// TIA Portal V17 export
FUNCTION "fcAllarmiTest" : Void   // FC195, LAD
{ S7_Optimized_Access := 'TRUE' }
// stored: SetENOAutomatically false
BEGIN

REGION Network 1: Alm200 - CB01: Timeout marcia avanti motore
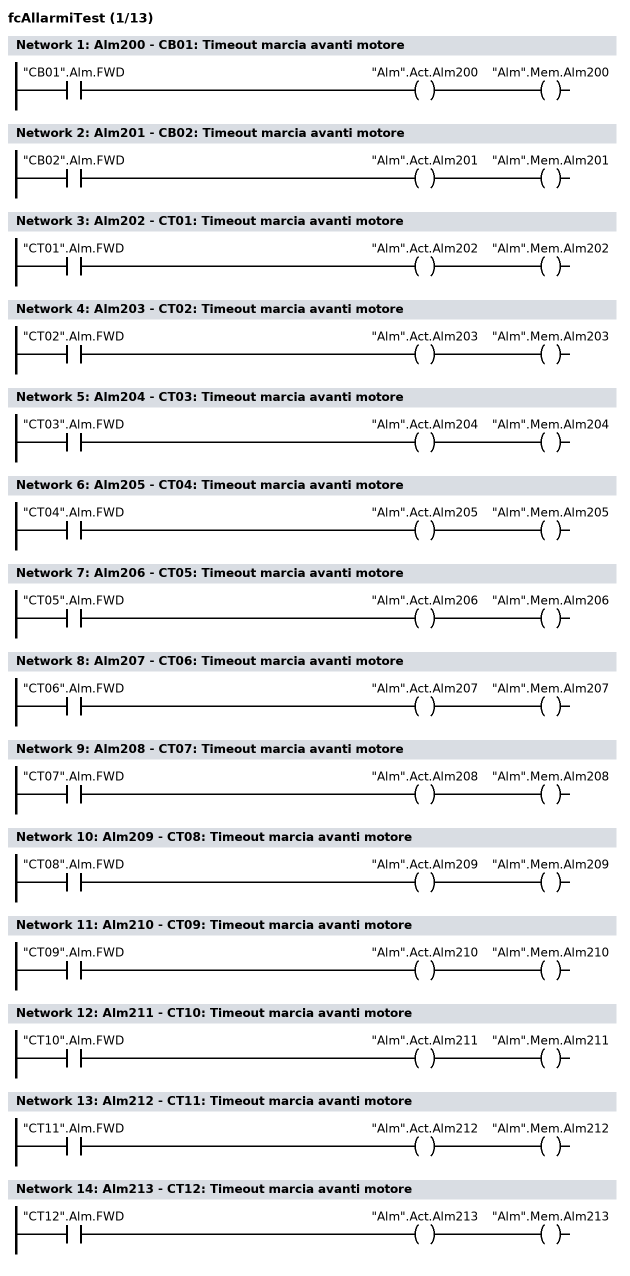
   RUNG wire#powerrail
      Contact( "CB01".Alm.FWD )
      Coil( "Alm".Act.Alm200 )
      Coil( "Alm".Mem.Alm200 )
   END_RUNG
   // the same network as SCL:
   "Alm".Act.Alm200 := "CB01".Alm.FWD;
   "Alm".Mem.Alm200 := "CB01".Alm.FWD;
END_REGION

REGION Network 2: Alm201 - CB02: Timeout marcia avanti motore
   RUNG wire#powerrail
      Contact( "CB02".Alm.FWD )
      Coil( "Alm".Act.Alm201 )
      Coil( "Alm".Mem.Alm201 )
   END_RUNG
   // the same network as SCL:
   "Alm".Act.Alm201 := "CB02".Alm.FWD;
   "Alm".Mem.Alm201 := "CB02".Alm.FWD;
END_REGION

REGION Network 3: Alm202 - CT01: Timeout marcia avanti motore
   RUNG wire#powerrail
      Contact( "CT01".Alm.FWD )
      Coil( "Alm".Act.Alm202 )
      Coil( "Alm".Mem.Alm202 )
   END_RUNG
   // the same network as SCL:
   "Alm".Act.Alm202 := "CT01".Alm.FWD;
   "Alm".Mem.Alm202 := "CT01".Alm.FWD;
END_REGION

REGION Network 4: Alm203 - CT02: Timeout marcia avanti motore
   RUNG wire#powerrail
      Contact( "CT02".Alm.FWD )
      Coil( "Alm".Act.Alm203 )
      Coil( "Alm".Mem.Alm203 )
   END_RUNG
   // the same network as SCL:
   "Alm".Act.Alm203 := "CT02".Alm.FWD;
   "Alm".Mem.Alm203 := "CT02".Alm.FWD;
END_REGION

REGION Network 5: Alm204 - CT03: Timeout marcia avanti motore
   RUNG wire#powerrail
      Contact( "CT03".Alm.FWD )
      Coil( "Alm".Act.Alm204 )
      Coil( "Alm".Mem.Alm204 )
   END_RUNG
   // the same network as SCL:
   "Alm".Act.Alm204 := "CT03".Alm.FWD;
   "Alm".Mem.Alm204 := "CT03".Alm.FWD;
END_REGION

REGION Network 6: Alm205 - CT04: Timeout marcia avanti motore
   RUNG wire#powerrail
      Contact( "CT04".Alm.FWD )
      Coil( "Alm".Act.Alm205 )
      Coil( "Alm".Mem.Alm205 )
   END_RUNG
   // the same network as SCL:
   "Alm".Act.Alm205 := "CT04".Alm.FWD;
   "Alm".Mem.Alm205 := "CT04".Alm.FWD;
END_REGION

REGION Network 7: Alm206 - CT05: Timeout marcia avanti motore
   RUNG wire#powerrail
      Contact( "CT05".Alm.FWD )
      Coil( "Alm".Act.Alm206 )
      Coil( "Alm".Mem.Alm206 )
   END_RUNG
   // the same network as SCL:
   "Alm".Act.Alm206 := "CT05".Alm.FWD;
   "Alm".Mem.Alm206 := "CT05".Alm.FWD;
END_REGION

REGION Network 8: Alm207 - CT06: Timeout marcia avanti motore
   RUNG wire#powerrail
      Contact( "CT06".Alm.FWD )
      Coil( "Alm".Act.Alm207 )
      Coil( "Alm".Mem.Alm207 )
   END_RUNG
   // the same network as SCL:
   "Alm".Act.Alm207 := "CT06".Alm.FWD;
   "Alm".Mem.Alm207 := "CT06".Alm.FWD;
END_REGION

REGION Network 9: Alm208 - CT07: Timeout marcia avanti motore
   RUNG wire#powerrail
      Contact( "CT07".Alm.FWD )
      Coil( "Alm".Act.Alm208 )
      Coil( "Alm".Mem.Alm208 )
   END_RUNG
   // the same network as SCL:
   "Alm".Act.Alm208 := "CT07".Alm.FWD;
   "Alm".Mem.Alm208 := "CT07".Alm.FWD;
END_REGION

REGION Network 10: Alm209 - CT08: Timeout marcia avanti motore
   RUNG wire#powerrail
      Contact( "CT08".Alm.FWD )
      Coil( "Alm".Act.Alm209 )
      Coil( "Alm".Mem.Alm209 )
   END_RUNG
   // the same network as SCL:
   "Alm".Act.Alm209 := "CT08".Alm.FWD;
   "Alm".Mem.Alm209 := "CT08".Alm.FWD;
END_REGION

REGION Network 11: Alm210 - CT09: Timeout marcia avanti motore
   RUNG wire#powerrail
      Contact( "CT09".Alm.FWD )
      Coil( "Alm".Act.Alm210 )
      Coil( "Alm".Mem.Alm210 )
   END_RUNG
   // the same network as SCL:
   "Alm".Act.Alm210 := "CT09".Alm.FWD;
   "Alm".Mem.Alm210 := "CT09".Alm.FWD;
END_REGION

REGION Network 12: Alm211 - CT10: Timeout marcia avanti motore
   RUNG wire#powerrail
      Contact( "CT10".Alm.FWD )
      Coil( "Alm".Act.Alm211 )
      Coil( "Alm".Mem.Alm211 )
   END_RUNG
   // the same network as SCL:
   "Alm".Act.Alm211 := "CT10".Alm.FWD;
   "Alm".Mem.Alm211 := "CT10".Alm.FWD;
END_REGION

REGION Network 13: Alm212 - CT11: Timeout marcia avanti motore
   RUNG wire#powerrail
      Contact( "CT11".Alm.FWD )
      Coil( "Alm".Act.Alm212 )
      Coil( "Alm".Mem.Alm212 )
   END_RUNG
   // the same network as SCL:
   "Alm".Act.Alm212 := "CT11".Alm.FWD;
   "Alm".Mem.Alm212 := "CT11".Alm.FWD;
END_REGION

REGION Network 14: Alm213 - CT12: Timeout marcia avanti motore
   RUNG wire#powerrail
      Contact( "CT12".Alm.FWD )
      Coil( "Alm".Act.Alm213 )
      Coil( "Alm".Mem.Alm213 )
   END_RUNG
   // the same network as SCL:
   "Alm".Act.Alm213 := "CT12".Alm.FWD;
   "Alm".Mem.Alm213 := "CT12".Alm.FWD;
END_REGION

REGION Network 15: Alm214 - CT13: Timeout marcia avanti motore
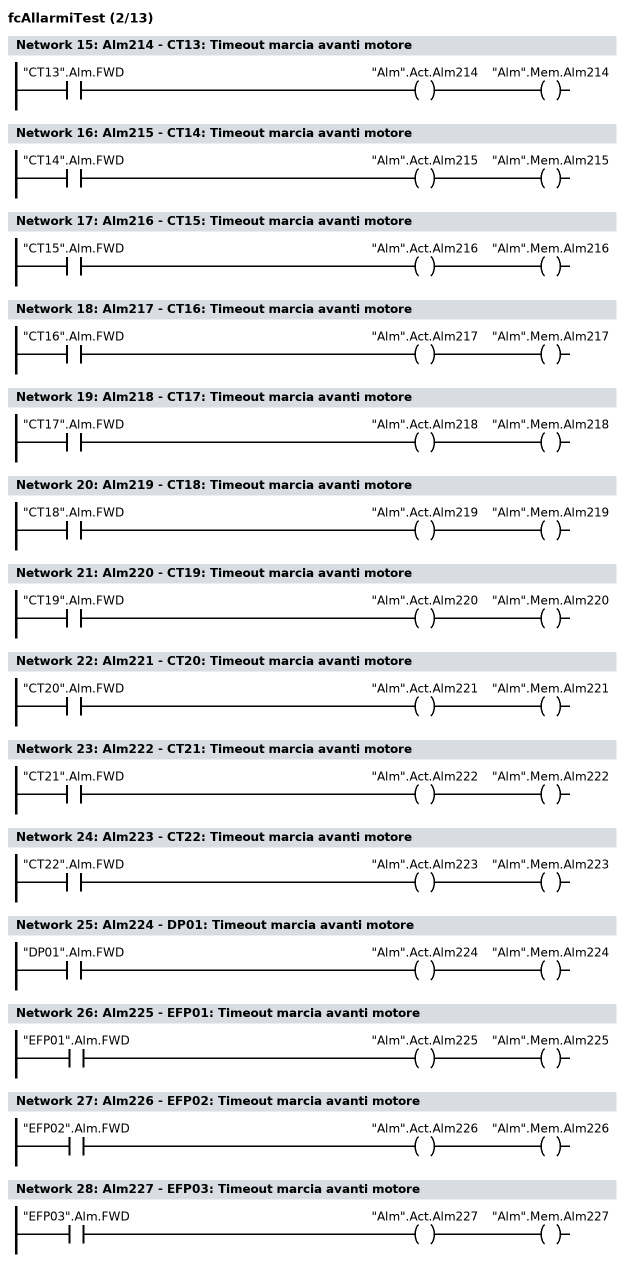
   RUNG wire#powerrail
      Contact( "CT13".Alm.FWD )
      Coil( "Alm".Act.Alm214 )
      Coil( "Alm".Mem.Alm214 )
   END_RUNG
   // the same network as SCL:
   "Alm".Act.Alm214 := "CT13".Alm.FWD;
   "Alm".Mem.Alm214 := "CT13".Alm.FWD;
END_REGION

REGION Network 16: Alm215 - CT14: Timeout marcia avanti motore
   RUNG wire#powerrail
      Contact( "CT14".Alm.FWD )
      Coil( "Alm".Act.Alm215 )
      Coil( "Alm".Mem.Alm215 )
   END_RUNG
   // the same network as SCL:
   "Alm".Act.Alm215 := "CT14".Alm.FWD;
   "Alm".Mem.Alm215 := "CT14".Alm.FWD;
END_REGION

REGION Network 17: Alm216 - CT15: Timeout marcia avanti motore
   RUNG wire#powerrail
      Contact( "CT15".Alm.FWD )
      Coil( "Alm".Act.Alm216 )
      Coil( "Alm".Mem.Alm216 )
   END_RUNG
   // the same network as SCL:
   "Alm".Act.Alm216 := "CT15".Alm.FWD;
   "Alm".Mem.Alm216 := "CT15".Alm.FWD;
END_REGION

REGION Network 18: Alm217 - CT16: Timeout marcia avanti motore
   RUNG wire#powerrail
      Contact( "CT16".Alm.FWD )
      Coil( "Alm".Act.Alm217 )
      Coil( "Alm".Mem.Alm217 )
   END_RUNG
   // the same network as SCL:
   "Alm".Act.Alm217 := "CT16".Alm.FWD;
   "Alm".Mem.Alm217 := "CT16".Alm.FWD;
END_REGION

REGION Network 19: Alm218 - CT17: Timeout marcia avanti motore
   RUNG wire#powerrail
      Contact( "CT17".Alm.FWD )
      Coil( "Alm".Act.Alm218 )
      Coil( "Alm".Mem.Alm218 )
   END_RUNG
   // the same network as SCL:
   "Alm".Act.Alm218 := "CT17".Alm.FWD;
   "Alm".Mem.Alm218 := "CT17".Alm.FWD;
END_REGION

REGION Network 20: Alm219 - CT18: Timeout marcia avanti motore
   RUNG wire#powerrail
      Contact( "CT18".Alm.FWD )
      Coil( "Alm".Act.Alm219 )
      Coil( "Alm".Mem.Alm219 )
   END_RUNG
   // the same network as SCL:
   "Alm".Act.Alm219 := "CT18".Alm.FWD;
   "Alm".Mem.Alm219 := "CT18".Alm.FWD;
END_REGION

REGION Network 21: Alm220 - CT19: Timeout marcia avanti motore
   RUNG wire#powerrail
      Contact( "CT19".Alm.FWD )
      Coil( "Alm".Act.Alm220 )
      Coil( "Alm".Mem.Alm220 )
   END_RUNG
   // the same network as SCL:
   "Alm".Act.Alm220 := "CT19".Alm.FWD;
   "Alm".Mem.Alm220 := "CT19".Alm.FWD;
END_REGION

REGION Network 22: Alm221 - CT20: Timeout marcia avanti motore
   RUNG wire#powerrail
      Contact( "CT20".Alm.FWD )
      Coil( "Alm".Act.Alm221 )
      Coil( "Alm".Mem.Alm221 )
   END_RUNG
   // the same network as SCL:
   "Alm".Act.Alm221 := "CT20".Alm.FWD;
   "Alm".Mem.Alm221 := "CT20".Alm.FWD;
END_REGION

REGION Network 23: Alm222 - CT21: Timeout marcia avanti motore
   RUNG wire#powerrail
      Contact( "CT21".Alm.FWD )
      Coil( "Alm".Act.Alm222 )
      Coil( "Alm".Mem.Alm222 )
   END_RUNG
   // the same network as SCL:
   "Alm".Act.Alm222 := "CT21".Alm.FWD;
   "Alm".Mem.Alm222 := "CT21".Alm.FWD;
END_REGION

REGION Network 24: Alm223 - CT22: Timeout marcia avanti motore
   RUNG wire#powerrail
      Contact( "CT22".Alm.FWD )
      Coil( "Alm".Act.Alm223 )
      Coil( "Alm".Mem.Alm223 )
   END_RUNG
   // the same network as SCL:
   "Alm".Act.Alm223 := "CT22".Alm.FWD;
   "Alm".Mem.Alm223 := "CT22".Alm.FWD;
END_REGION

REGION Network 25: Alm224 - DP01: Timeout marcia avanti motore
   RUNG wire#powerrail
      Contact( "DP01".Alm.FWD )
      Coil( "Alm".Act.Alm224 )
      Coil( "Alm".Mem.Alm224 )
   END_RUNG
   // the same network as SCL:
   "Alm".Act.Alm224 := "DP01".Alm.FWD;
   "Alm".Mem.Alm224 := "DP01".Alm.FWD;
END_REGION

REGION Network 26: Alm225 - EFP01: Timeout marcia avanti motore
   RUNG wire#powerrail
      Contact( "EFP01".Alm.FWD )
      Coil( "Alm".Act.Alm225 )
      Coil( "Alm".Mem.Alm225 )
   END_RUNG
   // the same network as SCL:
   "Alm".Act.Alm225 := "EFP01".Alm.FWD;
   "Alm".Mem.Alm225 := "EFP01".Alm.FWD;
END_REGION

REGION Network 27: Alm226 - EFP02: Timeout marcia avanti motore
   RUNG wire#powerrail
      Contact( "EFP02".Alm.FWD )
      Coil( "Alm".Act.Alm226 )
      Coil( "Alm".Mem.Alm226 )
   END_RUNG
   // the same network as SCL:
   "Alm".Act.Alm226 := "EFP02".Alm.FWD;
   "Alm".Mem.Alm226 := "EFP02".Alm.FWD;
END_REGION

REGION Network 28: Alm227 - EFP03: Timeout marcia avanti motore
   RUNG wire#powerrail
      Contact( "EFP03".Alm.FWD )
      Coil( "Alm".Act.Alm227 )
      Coil( "Alm".Mem.Alm227 )
   END_RUNG
   // the same network as SCL:
   "Alm".Act.Alm227 := "EFP03".Alm.FWD;
   "Alm".Mem.Alm227 := "EFP03".Alm.FWD;
END_REGION

REGION Network 29: Alm228 - EFP04: Timeout marcia avanti motore
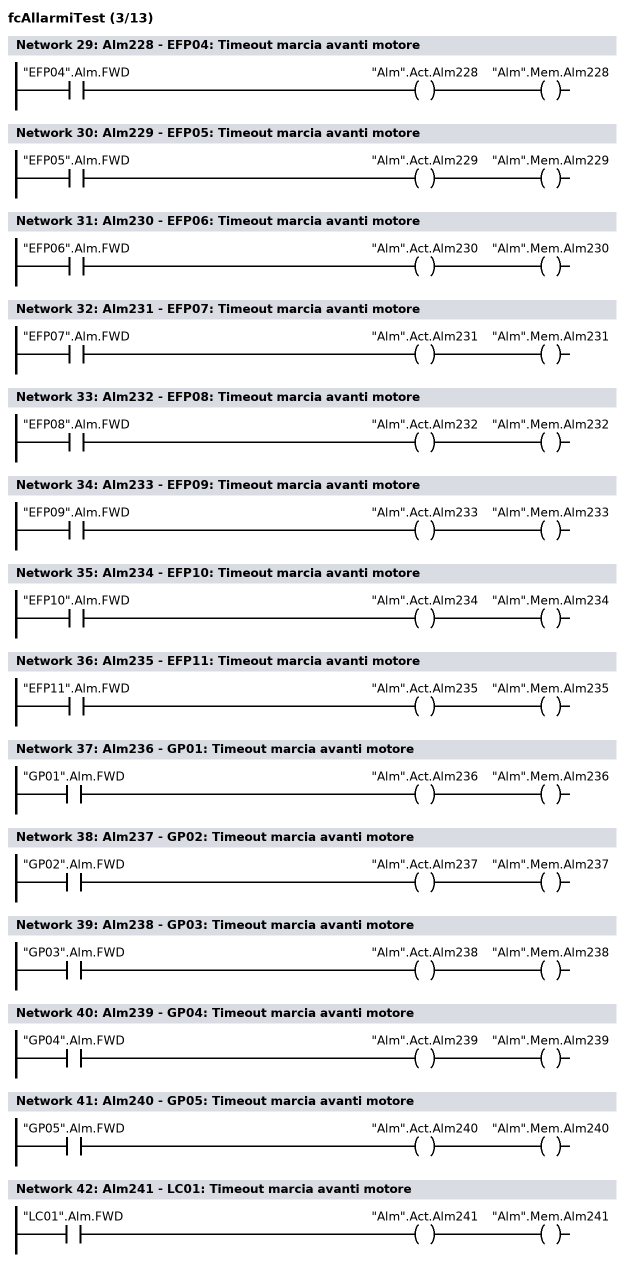
   RUNG wire#powerrail
      Contact( "EFP04".Alm.FWD )
      Coil( "Alm".Act.Alm228 )
      Coil( "Alm".Mem.Alm228 )
   END_RUNG
   // the same network as SCL:
   "Alm".Act.Alm228 := "EFP04".Alm.FWD;
   "Alm".Mem.Alm228 := "EFP04".Alm.FWD;
END_REGION

REGION Network 30: Alm229 - EFP05: Timeout marcia avanti motore
   RUNG wire#powerrail
      Contact( "EFP05".Alm.FWD )
      Coil( "Alm".Act.Alm229 )
      Coil( "Alm".Mem.Alm229 )
   END_RUNG
   // the same network as SCL:
   "Alm".Act.Alm229 := "EFP05".Alm.FWD;
   "Alm".Mem.Alm229 := "EFP05".Alm.FWD;
END_REGION

REGION Network 31: Alm230 - EFP06: Timeout marcia avanti motore
   RUNG wire#powerrail
      Contact( "EFP06".Alm.FWD )
      Coil( "Alm".Act.Alm230 )
      Coil( "Alm".Mem.Alm230 )
   END_RUNG
   // the same network as SCL:
   "Alm".Act.Alm230 := "EFP06".Alm.FWD;
   "Alm".Mem.Alm230 := "EFP06".Alm.FWD;
END_REGION

REGION Network 32: Alm231 - EFP07: Timeout marcia avanti motore
   RUNG wire#powerrail
      Contact( "EFP07".Alm.FWD )
      Coil( "Alm".Act.Alm231 )
      Coil( "Alm".Mem.Alm231 )
   END_RUNG
   // the same network as SCL:
   "Alm".Act.Alm231 := "EFP07".Alm.FWD;
   "Alm".Mem.Alm231 := "EFP07".Alm.FWD;
END_REGION

REGION Network 33: Alm232 - EFP08: Timeout marcia avanti motore
   RUNG wire#powerrail
      Contact( "EFP08".Alm.FWD )
      Coil( "Alm".Act.Alm232 )
      Coil( "Alm".Mem.Alm232 )
   END_RUNG
   // the same network as SCL:
   "Alm".Act.Alm232 := "EFP08".Alm.FWD;
   "Alm".Mem.Alm232 := "EFP08".Alm.FWD;
END_REGION

REGION Network 34: Alm233 - EFP09: Timeout marcia avanti motore
   RUNG wire#powerrail
      Contact( "EFP09".Alm.FWD )
      Coil( "Alm".Act.Alm233 )
      Coil( "Alm".Mem.Alm233 )
   END_RUNG
   // the same network as SCL:
   "Alm".Act.Alm233 := "EFP09".Alm.FWD;
   "Alm".Mem.Alm233 := "EFP09".Alm.FWD;
END_REGION

REGION Network 35: Alm234 - EFP10: Timeout marcia avanti motore
   RUNG wire#powerrail
      Contact( "EFP10".Alm.FWD )
      Coil( "Alm".Act.Alm234 )
      Coil( "Alm".Mem.Alm234 )
   END_RUNG
   // the same network as SCL:
   "Alm".Act.Alm234 := "EFP10".Alm.FWD;
   "Alm".Mem.Alm234 := "EFP10".Alm.FWD;
END_REGION

REGION Network 36: Alm235 - EFP11: Timeout marcia avanti motore
   RUNG wire#powerrail
      Contact( "EFP11".Alm.FWD )
      Coil( "Alm".Act.Alm235 )
      Coil( "Alm".Mem.Alm235 )
   END_RUNG
   // the same network as SCL:
   "Alm".Act.Alm235 := "EFP11".Alm.FWD;
   "Alm".Mem.Alm235 := "EFP11".Alm.FWD;
END_REGION

REGION Network 37: Alm236 - GP01: Timeout marcia avanti motore
   RUNG wire#powerrail
      Contact( "GP01".Alm.FWD )
      Coil( "Alm".Act.Alm236 )
      Coil( "Alm".Mem.Alm236 )
   END_RUNG
   // the same network as SCL:
   "Alm".Act.Alm236 := "GP01".Alm.FWD;
   "Alm".Mem.Alm236 := "GP01".Alm.FWD;
END_REGION

REGION Network 38: Alm237 - GP02: Timeout marcia avanti motore
   RUNG wire#powerrail
      Contact( "GP02".Alm.FWD )
      Coil( "Alm".Act.Alm237 )
      Coil( "Alm".Mem.Alm237 )
   END_RUNG
   // the same network as SCL:
   "Alm".Act.Alm237 := "GP02".Alm.FWD;
   "Alm".Mem.Alm237 := "GP02".Alm.FWD;
END_REGION

REGION Network 39: Alm238 - GP03: Timeout marcia avanti motore
   RUNG wire#powerrail
      Contact( "GP03".Alm.FWD )
      Coil( "Alm".Act.Alm238 )
      Coil( "Alm".Mem.Alm238 )
   END_RUNG
   // the same network as SCL:
   "Alm".Act.Alm238 := "GP03".Alm.FWD;
   "Alm".Mem.Alm238 := "GP03".Alm.FWD;
END_REGION

REGION Network 40: Alm239 - GP04: Timeout marcia avanti motore
   RUNG wire#powerrail
      Contact( "GP04".Alm.FWD )
      Coil( "Alm".Act.Alm239 )
      Coil( "Alm".Mem.Alm239 )
   END_RUNG
   // the same network as SCL:
   "Alm".Act.Alm239 := "GP04".Alm.FWD;
   "Alm".Mem.Alm239 := "GP04".Alm.FWD;
END_REGION

REGION Network 41: Alm240 - GP05: Timeout marcia avanti motore
   RUNG wire#powerrail
      Contact( "GP05".Alm.FWD )
      Coil( "Alm".Act.Alm240 )
      Coil( "Alm".Mem.Alm240 )
   END_RUNG
   // the same network as SCL:
   "Alm".Act.Alm240 := "GP05".Alm.FWD;
   "Alm".Mem.Alm240 := "GP05".Alm.FWD;
END_REGION

REGION Network 42: Alm241 - LC01: Timeout marcia avanti motore
   RUNG wire#powerrail
      Contact( "LC01".Alm.FWD )
      Coil( "Alm".Act.Alm241 )
      Coil( "Alm".Mem.Alm241 )
   END_RUNG
   // the same network as SCL:
   "Alm".Act.Alm241 := "LC01".Alm.FWD;
   "Alm".Mem.Alm241 := "LC01".Alm.FWD;
END_REGION

REGION Network 43: Alm242 - LC02: Timeout marcia avanti motore
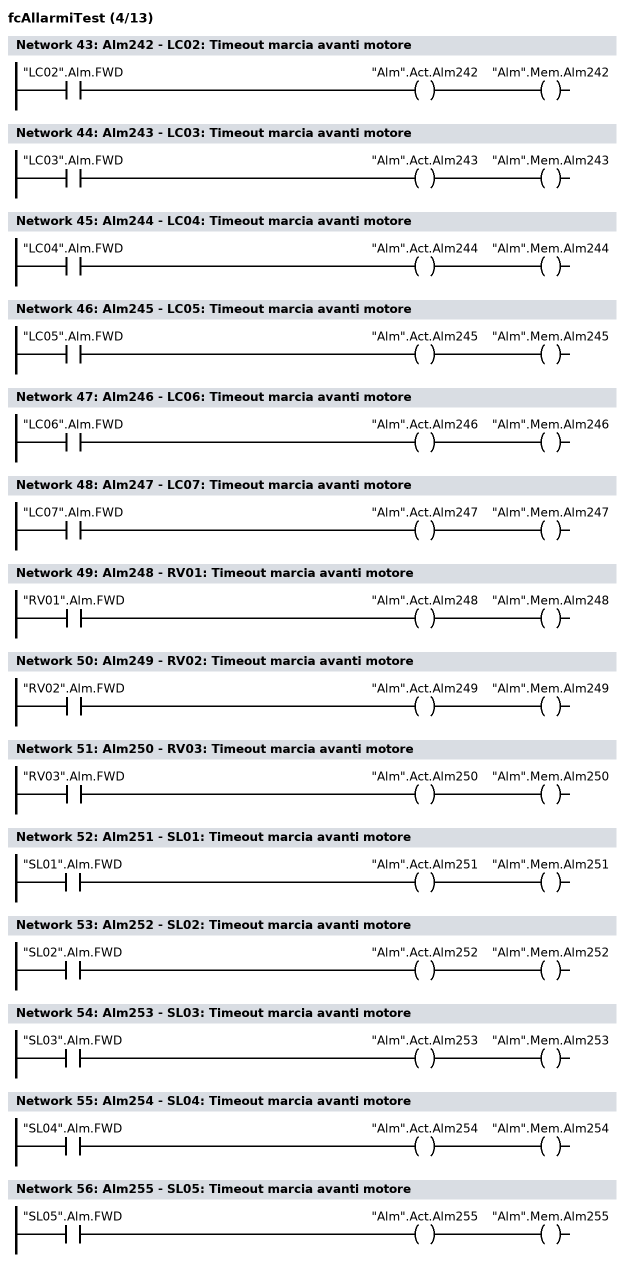
   RUNG wire#powerrail
      Contact( "LC02".Alm.FWD )
      Coil( "Alm".Act.Alm242 )
      Coil( "Alm".Mem.Alm242 )
   END_RUNG
   // the same network as SCL:
   "Alm".Act.Alm242 := "LC02".Alm.FWD;
   "Alm".Mem.Alm242 := "LC02".Alm.FWD;
END_REGION

REGION Network 44: Alm243 - LC03: Timeout marcia avanti motore
   RUNG wire#powerrail
      Contact( "LC03".Alm.FWD )
      Coil( "Alm".Act.Alm243 )
      Coil( "Alm".Mem.Alm243 )
   END_RUNG
   // the same network as SCL:
   "Alm".Act.Alm243 := "LC03".Alm.FWD;
   "Alm".Mem.Alm243 := "LC03".Alm.FWD;
END_REGION

REGION Network 45: Alm244 - LC04: Timeout marcia avanti motore
   RUNG wire#powerrail
      Contact( "LC04".Alm.FWD )
      Coil( "Alm".Act.Alm244 )
      Coil( "Alm".Mem.Alm244 )
   END_RUNG
   // the same network as SCL:
   "Alm".Act.Alm244 := "LC04".Alm.FWD;
   "Alm".Mem.Alm244 := "LC04".Alm.FWD;
END_REGION

REGION Network 46: Alm245 - LC05: Timeout marcia avanti motore
   RUNG wire#powerrail
      Contact( "LC05".Alm.FWD )
      Coil( "Alm".Act.Alm245 )
      Coil( "Alm".Mem.Alm245 )
   END_RUNG
   // the same network as SCL:
   "Alm".Act.Alm245 := "LC05".Alm.FWD;
   "Alm".Mem.Alm245 := "LC05".Alm.FWD;
END_REGION

REGION Network 47: Alm246 - LC06: Timeout marcia avanti motore
   RUNG wire#powerrail
      Contact( "LC06".Alm.FWD )
      Coil( "Alm".Act.Alm246 )
      Coil( "Alm".Mem.Alm246 )
   END_RUNG
   // the same network as SCL:
   "Alm".Act.Alm246 := "LC06".Alm.FWD;
   "Alm".Mem.Alm246 := "LC06".Alm.FWD;
END_REGION

REGION Network 48: Alm247 - LC07: Timeout marcia avanti motore
   RUNG wire#powerrail
      Contact( "LC07".Alm.FWD )
      Coil( "Alm".Act.Alm247 )
      Coil( "Alm".Mem.Alm247 )
   END_RUNG
   // the same network as SCL:
   "Alm".Act.Alm247 := "LC07".Alm.FWD;
   "Alm".Mem.Alm247 := "LC07".Alm.FWD;
END_REGION

REGION Network 49: Alm248 - RV01: Timeout marcia avanti motore
   RUNG wire#powerrail
      Contact( "RV01".Alm.FWD )
      Coil( "Alm".Act.Alm248 )
      Coil( "Alm".Mem.Alm248 )
   END_RUNG
   // the same network as SCL:
   "Alm".Act.Alm248 := "RV01".Alm.FWD;
   "Alm".Mem.Alm248 := "RV01".Alm.FWD;
END_REGION

REGION Network 50: Alm249 - RV02: Timeout marcia avanti motore
   RUNG wire#powerrail
      Contact( "RV02".Alm.FWD )
      Coil( "Alm".Act.Alm249 )
      Coil( "Alm".Mem.Alm249 )
   END_RUNG
   // the same network as SCL:
   "Alm".Act.Alm249 := "RV02".Alm.FWD;
   "Alm".Mem.Alm249 := "RV02".Alm.FWD;
END_REGION

REGION Network 51: Alm250 - RV03: Timeout marcia avanti motore
   RUNG wire#powerrail
      Contact( "RV03".Alm.FWD )
      Coil( "Alm".Act.Alm250 )
      Coil( "Alm".Mem.Alm250 )
   END_RUNG
   // the same network as SCL:
   "Alm".Act.Alm250 := "RV03".Alm.FWD;
   "Alm".Mem.Alm250 := "RV03".Alm.FWD;
END_REGION

REGION Network 52: Alm251 - SL01: Timeout marcia avanti motore
   RUNG wire#powerrail
      Contact( "SL01".Alm.FWD )
      Coil( "Alm".Act.Alm251 )
      Coil( "Alm".Mem.Alm251 )
   END_RUNG
   // the same network as SCL:
   "Alm".Act.Alm251 := "SL01".Alm.FWD;
   "Alm".Mem.Alm251 := "SL01".Alm.FWD;
END_REGION

REGION Network 53: Alm252 - SL02: Timeout marcia avanti motore
   RUNG wire#powerrail
      Contact( "SL02".Alm.FWD )
      Coil( "Alm".Act.Alm252 )
      Coil( "Alm".Mem.Alm252 )
   END_RUNG
   // the same network as SCL:
   "Alm".Act.Alm252 := "SL02".Alm.FWD;
   "Alm".Mem.Alm252 := "SL02".Alm.FWD;
END_REGION

REGION Network 54: Alm253 - SL03: Timeout marcia avanti motore
   RUNG wire#powerrail
      Contact( "SL03".Alm.FWD )
      Coil( "Alm".Act.Alm253 )
      Coil( "Alm".Mem.Alm253 )
   END_RUNG
   // the same network as SCL:
   "Alm".Act.Alm253 := "SL03".Alm.FWD;
   "Alm".Mem.Alm253 := "SL03".Alm.FWD;
END_REGION

REGION Network 55: Alm254 - SL04: Timeout marcia avanti motore
   RUNG wire#powerrail
      Contact( "SL04".Alm.FWD )
      Coil( "Alm".Act.Alm254 )
      Coil( "Alm".Mem.Alm254 )
   END_RUNG
   // the same network as SCL:
   "Alm".Act.Alm254 := "SL04".Alm.FWD;
   "Alm".Mem.Alm254 := "SL04".Alm.FWD;
END_REGION

REGION Network 56: Alm255 - SL05: Timeout marcia avanti motore
   RUNG wire#powerrail
      Contact( "SL05".Alm.FWD )
      Coil( "Alm".Act.Alm255 )
      Coil( "Alm".Mem.Alm255 )
   END_RUNG
   // the same network as SCL:
   "Alm".Act.Alm255 := "SL05".Alm.FWD;
   "Alm".Mem.Alm255 := "SL05".Alm.FWD;
END_REGION

REGION Network 57: Alm256 - SL06: Timeout marcia avanti motore
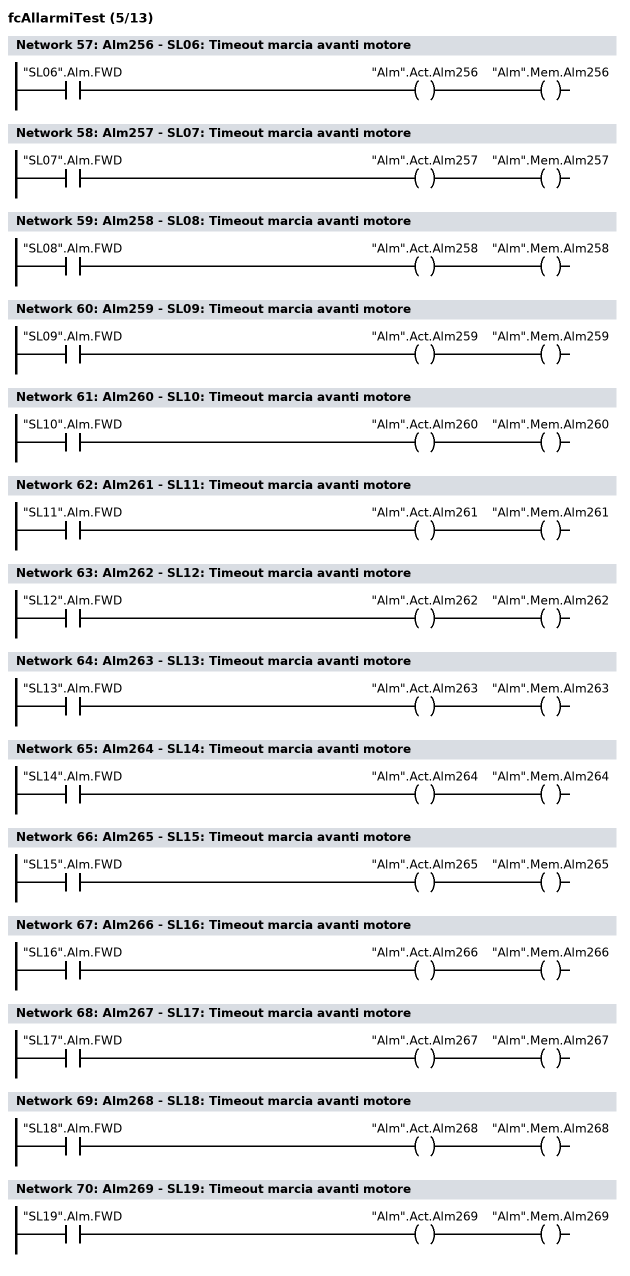
   RUNG wire#powerrail
      Contact( "SL06".Alm.FWD )
      Coil( "Alm".Act.Alm256 )
      Coil( "Alm".Mem.Alm256 )
   END_RUNG
   // the same network as SCL:
   "Alm".Act.Alm256 := "SL06".Alm.FWD;
   "Alm".Mem.Alm256 := "SL06".Alm.FWD;
END_REGION

REGION Network 58: Alm257 - SL07: Timeout marcia avanti motore
   RUNG wire#powerrail
      Contact( "SL07".Alm.FWD )
      Coil( "Alm".Act.Alm257 )
      Coil( "Alm".Mem.Alm257 )
   END_RUNG
   // the same network as SCL:
   "Alm".Act.Alm257 := "SL07".Alm.FWD;
   "Alm".Mem.Alm257 := "SL07".Alm.FWD;
END_REGION

REGION Network 59: Alm258 - SL08: Timeout marcia avanti motore
   RUNG wire#powerrail
      Contact( "SL08".Alm.FWD )
      Coil( "Alm".Act.Alm258 )
      Coil( "Alm".Mem.Alm258 )
   END_RUNG
   // the same network as SCL:
   "Alm".Act.Alm258 := "SL08".Alm.FWD;
   "Alm".Mem.Alm258 := "SL08".Alm.FWD;
END_REGION

REGION Network 60: Alm259 - SL09: Timeout marcia avanti motore
   RUNG wire#powerrail
      Contact( "SL09".Alm.FWD )
      Coil( "Alm".Act.Alm259 )
      Coil( "Alm".Mem.Alm259 )
   END_RUNG
   // the same network as SCL:
   "Alm".Act.Alm259 := "SL09".Alm.FWD;
   "Alm".Mem.Alm259 := "SL09".Alm.FWD;
END_REGION

REGION Network 61: Alm260 - SL10: Timeout marcia avanti motore
   RUNG wire#powerrail
      Contact( "SL10".Alm.FWD )
      Coil( "Alm".Act.Alm260 )
      Coil( "Alm".Mem.Alm260 )
   END_RUNG
   // the same network as SCL:
   "Alm".Act.Alm260 := "SL10".Alm.FWD;
   "Alm".Mem.Alm260 := "SL10".Alm.FWD;
END_REGION

REGION Network 62: Alm261 - SL11: Timeout marcia avanti motore
   RUNG wire#powerrail
      Contact( "SL11".Alm.FWD )
      Coil( "Alm".Act.Alm261 )
      Coil( "Alm".Mem.Alm261 )
   END_RUNG
   // the same network as SCL:
   "Alm".Act.Alm261 := "SL11".Alm.FWD;
   "Alm".Mem.Alm261 := "SL11".Alm.FWD;
END_REGION

REGION Network 63: Alm262 - SL12: Timeout marcia avanti motore
   RUNG wire#powerrail
      Contact( "SL12".Alm.FWD )
      Coil( "Alm".Act.Alm262 )
      Coil( "Alm".Mem.Alm262 )
   END_RUNG
   // the same network as SCL:
   "Alm".Act.Alm262 := "SL12".Alm.FWD;
   "Alm".Mem.Alm262 := "SL12".Alm.FWD;
END_REGION

REGION Network 64: Alm263 - SL13: Timeout marcia avanti motore
   RUNG wire#powerrail
      Contact( "SL13".Alm.FWD )
      Coil( "Alm".Act.Alm263 )
      Coil( "Alm".Mem.Alm263 )
   END_RUNG
   // the same network as SCL:
   "Alm".Act.Alm263 := "SL13".Alm.FWD;
   "Alm".Mem.Alm263 := "SL13".Alm.FWD;
END_REGION

REGION Network 65: Alm264 - SL14: Timeout marcia avanti motore
   RUNG wire#powerrail
      Contact( "SL14".Alm.FWD )
      Coil( "Alm".Act.Alm264 )
      Coil( "Alm".Mem.Alm264 )
   END_RUNG
   // the same network as SCL:
   "Alm".Act.Alm264 := "SL14".Alm.FWD;
   "Alm".Mem.Alm264 := "SL14".Alm.FWD;
END_REGION

REGION Network 66: Alm265 - SL15: Timeout marcia avanti motore
   RUNG wire#powerrail
      Contact( "SL15".Alm.FWD )
      Coil( "Alm".Act.Alm265 )
      Coil( "Alm".Mem.Alm265 )
   END_RUNG
   // the same network as SCL:
   "Alm".Act.Alm265 := "SL15".Alm.FWD;
   "Alm".Mem.Alm265 := "SL15".Alm.FWD;
END_REGION

REGION Network 67: Alm266 - SL16: Timeout marcia avanti motore
   RUNG wire#powerrail
      Contact( "SL16".Alm.FWD )
      Coil( "Alm".Act.Alm266 )
      Coil( "Alm".Mem.Alm266 )
   END_RUNG
   // the same network as SCL:
   "Alm".Act.Alm266 := "SL16".Alm.FWD;
   "Alm".Mem.Alm266 := "SL16".Alm.FWD;
END_REGION

REGION Network 68: Alm267 - SL17: Timeout marcia avanti motore
   RUNG wire#powerrail
      Contact( "SL17".Alm.FWD )
      Coil( "Alm".Act.Alm267 )
      Coil( "Alm".Mem.Alm267 )
   END_RUNG
   // the same network as SCL:
   "Alm".Act.Alm267 := "SL17".Alm.FWD;
   "Alm".Mem.Alm267 := "SL17".Alm.FWD;
END_REGION

REGION Network 69: Alm268 - SL18: Timeout marcia avanti motore
   RUNG wire#powerrail
      Contact( "SL18".Alm.FWD )
      Coil( "Alm".Act.Alm268 )
      Coil( "Alm".Mem.Alm268 )
   END_RUNG
   // the same network as SCL:
   "Alm".Act.Alm268 := "SL18".Alm.FWD;
   "Alm".Mem.Alm268 := "SL18".Alm.FWD;
END_REGION

REGION Network 70: Alm269 - SL19: Timeout marcia avanti motore
   RUNG wire#powerrail
      Contact( "SL19".Alm.FWD )
      Coil( "Alm".Act.Alm269 )
      Coil( "Alm".Mem.Alm269 )
   END_RUNG
   // the same network as SCL:
   "Alm".Act.Alm269 := "SL19".Alm.FWD;
   "Alm".Mem.Alm269 := "SL19".Alm.FWD;
END_REGION

REGION Network 71: Alm270 - SL20: Timeout marcia avanti motore
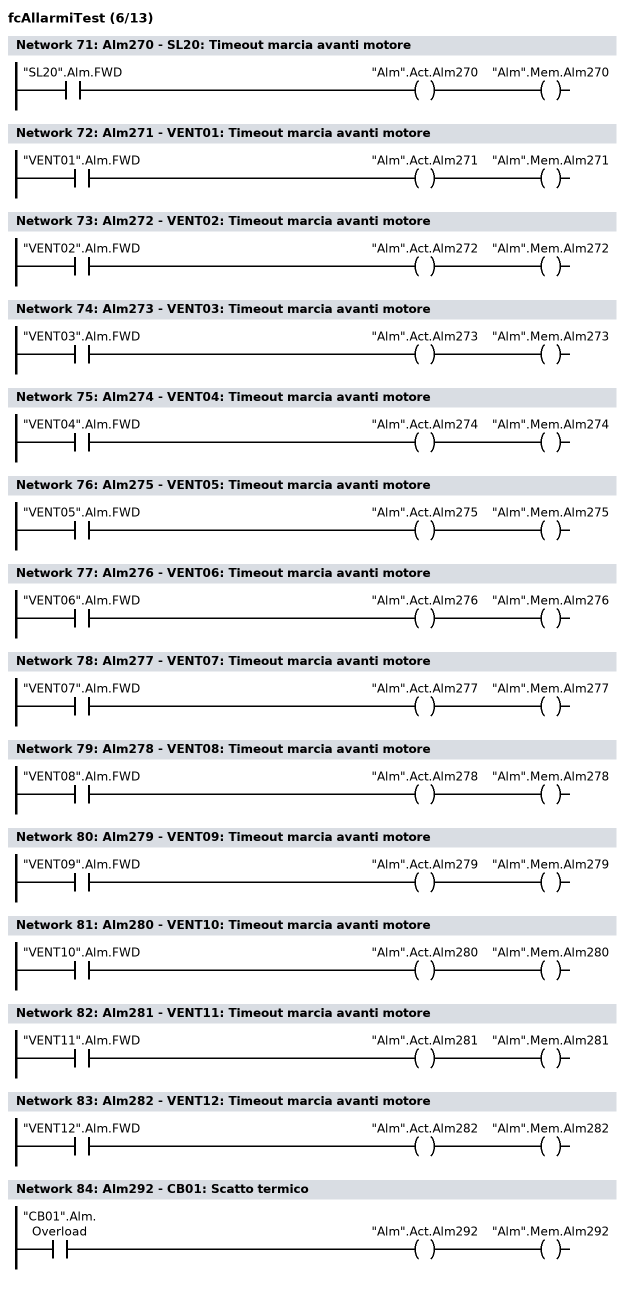
   RUNG wire#powerrail
      Contact( "SL20".Alm.FWD )
      Coil( "Alm".Act.Alm270 )
      Coil( "Alm".Mem.Alm270 )
   END_RUNG
   // the same network as SCL:
   "Alm".Act.Alm270 := "SL20".Alm.FWD;
   "Alm".Mem.Alm270 := "SL20".Alm.FWD;
END_REGION

REGION Network 72: Alm271 - VENT01: Timeout marcia avanti motore
   RUNG wire#powerrail
      Contact( "VENT01".Alm.FWD )
      Coil( "Alm".Act.Alm271 )
      Coil( "Alm".Mem.Alm271 )
   END_RUNG
   // the same network as SCL:
   "Alm".Act.Alm271 := "VENT01".Alm.FWD;
   "Alm".Mem.Alm271 := "VENT01".Alm.FWD;
END_REGION

REGION Network 73: Alm272 - VENT02: Timeout marcia avanti motore
   RUNG wire#powerrail
      Contact( "VENT02".Alm.FWD )
      Coil( "Alm".Act.Alm272 )
      Coil( "Alm".Mem.Alm272 )
   END_RUNG
   // the same network as SCL:
   "Alm".Act.Alm272 := "VENT02".Alm.FWD;
   "Alm".Mem.Alm272 := "VENT02".Alm.FWD;
END_REGION

REGION Network 74: Alm273 - VENT03: Timeout marcia avanti motore
   RUNG wire#powerrail
      Contact( "VENT03".Alm.FWD )
      Coil( "Alm".Act.Alm273 )
      Coil( "Alm".Mem.Alm273 )
   END_RUNG
   // the same network as SCL:
   "Alm".Act.Alm273 := "VENT03".Alm.FWD;
   "Alm".Mem.Alm273 := "VENT03".Alm.FWD;
END_REGION

REGION Network 75: Alm274 - VENT04: Timeout marcia avanti motore
   RUNG wire#powerrail
      Contact( "VENT04".Alm.FWD )
      Coil( "Alm".Act.Alm274 )
      Coil( "Alm".Mem.Alm274 )
   END_RUNG
   // the same network as SCL:
   "Alm".Act.Alm274 := "VENT04".Alm.FWD;
   "Alm".Mem.Alm274 := "VENT04".Alm.FWD;
END_REGION

REGION Network 76: Alm275 - VENT05: Timeout marcia avanti motore
   RUNG wire#powerrail
      Contact( "VENT05".Alm.FWD )
      Coil( "Alm".Act.Alm275 )
      Coil( "Alm".Mem.Alm275 )
   END_RUNG
   // the same network as SCL:
   "Alm".Act.Alm275 := "VENT05".Alm.FWD;
   "Alm".Mem.Alm275 := "VENT05".Alm.FWD;
END_REGION

REGION Network 77: Alm276 - VENT06: Timeout marcia avanti motore
   RUNG wire#powerrail
      Contact( "VENT06".Alm.FWD )
      Coil( "Alm".Act.Alm276 )
      Coil( "Alm".Mem.Alm276 )
   END_RUNG
   // the same network as SCL:
   "Alm".Act.Alm276 := "VENT06".Alm.FWD;
   "Alm".Mem.Alm276 := "VENT06".Alm.FWD;
END_REGION

REGION Network 78: Alm277 - VENT07: Timeout marcia avanti motore
   RUNG wire#powerrail
      Contact( "VENT07".Alm.FWD )
      Coil( "Alm".Act.Alm277 )
      Coil( "Alm".Mem.Alm277 )
   END_RUNG
   // the same network as SCL:
   "Alm".Act.Alm277 := "VENT07".Alm.FWD;
   "Alm".Mem.Alm277 := "VENT07".Alm.FWD;
END_REGION

REGION Network 79: Alm278 - VENT08: Timeout marcia avanti motore
   RUNG wire#powerrail
      Contact( "VENT08".Alm.FWD )
      Coil( "Alm".Act.Alm278 )
      Coil( "Alm".Mem.Alm278 )
   END_RUNG
   // the same network as SCL:
   "Alm".Act.Alm278 := "VENT08".Alm.FWD;
   "Alm".Mem.Alm278 := "VENT08".Alm.FWD;
END_REGION

REGION Network 80: Alm279 - VENT09: Timeout marcia avanti motore
   RUNG wire#powerrail
      Contact( "VENT09".Alm.FWD )
      Coil( "Alm".Act.Alm279 )
      Coil( "Alm".Mem.Alm279 )
   END_RUNG
   // the same network as SCL:
   "Alm".Act.Alm279 := "VENT09".Alm.FWD;
   "Alm".Mem.Alm279 := "VENT09".Alm.FWD;
END_REGION

REGION Network 81: Alm280 - VENT10: Timeout marcia avanti motore
   RUNG wire#powerrail
      Contact( "VENT10".Alm.FWD )
      Coil( "Alm".Act.Alm280 )
      Coil( "Alm".Mem.Alm280 )
   END_RUNG
   // the same network as SCL:
   "Alm".Act.Alm280 := "VENT10".Alm.FWD;
   "Alm".Mem.Alm280 := "VENT10".Alm.FWD;
END_REGION

REGION Network 82: Alm281 - VENT11: Timeout marcia avanti motore
   RUNG wire#powerrail
      Contact( "VENT11".Alm.FWD )
      Coil( "Alm".Act.Alm281 )
      Coil( "Alm".Mem.Alm281 )
   END_RUNG
   // the same network as SCL:
   "Alm".Act.Alm281 := "VENT11".Alm.FWD;
   "Alm".Mem.Alm281 := "VENT11".Alm.FWD;
END_REGION

REGION Network 83: Alm282 - VENT12: Timeout marcia avanti motore
   RUNG wire#powerrail
      Contact( "VENT12".Alm.FWD )
      Coil( "Alm".Act.Alm282 )
      Coil( "Alm".Mem.Alm282 )
   END_RUNG
   // the same network as SCL:
   "Alm".Act.Alm282 := "VENT12".Alm.FWD;
   "Alm".Mem.Alm282 := "VENT12".Alm.FWD;
END_REGION

REGION Network 84: Alm292 - CB01: Scatto termico
   RUNG wire#powerrail
      Contact( "CB01".Alm.Overload )
      Coil( "Alm".Act.Alm292 )
      Coil( "Alm".Mem.Alm292 )
   END_RUNG
   // the same network as SCL:
   "Alm".Act.Alm292 := "CB01".Alm.Overload;
   "Alm".Mem.Alm292 := "CB01".Alm.Overload;
END_REGION

REGION Network 85: Alm293 - CB02: Scatto termico
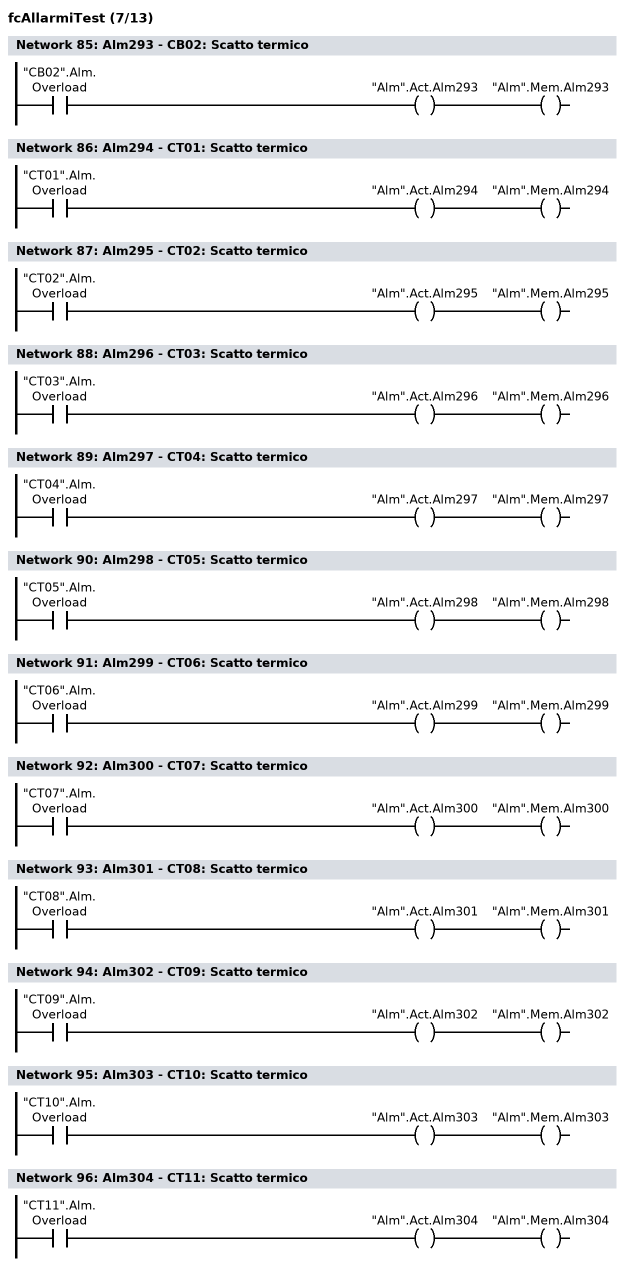
   RUNG wire#powerrail
      Contact( "CB02".Alm.Overload )
      Coil( "Alm".Act.Alm293 )
      Coil( "Alm".Mem.Alm293 )
   END_RUNG
   // the same network as SCL:
   "Alm".Act.Alm293 := "CB02".Alm.Overload;
   "Alm".Mem.Alm293 := "CB02".Alm.Overload;
END_REGION

REGION Network 86: Alm294 - CT01: Scatto termico
   RUNG wire#powerrail
      Contact( "CT01".Alm.Overload )
      Coil( "Alm".Act.Alm294 )
      Coil( "Alm".Mem.Alm294 )
   END_RUNG
   // the same network as SCL:
   "Alm".Act.Alm294 := "CT01".Alm.Overload;
   "Alm".Mem.Alm294 := "CT01".Alm.Overload;
END_REGION

REGION Network 87: Alm295 - CT02: Scatto termico
   RUNG wire#powerrail
      Contact( "CT02".Alm.Overload )
      Coil( "Alm".Act.Alm295 )
      Coil( "Alm".Mem.Alm295 )
   END_RUNG
   // the same network as SCL:
   "Alm".Act.Alm295 := "CT02".Alm.Overload;
   "Alm".Mem.Alm295 := "CT02".Alm.Overload;
END_REGION

REGION Network 88: Alm296 - CT03: Scatto termico
   RUNG wire#powerrail
      Contact( "CT03".Alm.Overload )
      Coil( "Alm".Act.Alm296 )
      Coil( "Alm".Mem.Alm296 )
   END_RUNG
   // the same network as SCL:
   "Alm".Act.Alm296 := "CT03".Alm.Overload;
   "Alm".Mem.Alm296 := "CT03".Alm.Overload;
END_REGION

REGION Network 89: Alm297 - CT04: Scatto termico
   RUNG wire#powerrail
      Contact( "CT04".Alm.Overload )
      Coil( "Alm".Act.Alm297 )
      Coil( "Alm".Mem.Alm297 )
   END_RUNG
   // the same network as SCL:
   "Alm".Act.Alm297 := "CT04".Alm.Overload;
   "Alm".Mem.Alm297 := "CT04".Alm.Overload;
END_REGION

REGION Network 90: Alm298 - CT05: Scatto termico
   RUNG wire#powerrail
      Contact( "CT05".Alm.Overload )
      Coil( "Alm".Act.Alm298 )
      Coil( "Alm".Mem.Alm298 )
   END_RUNG
   // the same network as SCL:
   "Alm".Act.Alm298 := "CT05".Alm.Overload;
   "Alm".Mem.Alm298 := "CT05".Alm.Overload;
END_REGION

REGION Network 91: Alm299 - CT06: Scatto termico
   RUNG wire#powerrail
      Contact( "CT06".Alm.Overload )
      Coil( "Alm".Act.Alm299 )
      Coil( "Alm".Mem.Alm299 )
   END_RUNG
   // the same network as SCL:
   "Alm".Act.Alm299 := "CT06".Alm.Overload;
   "Alm".Mem.Alm299 := "CT06".Alm.Overload;
END_REGION

REGION Network 92: Alm300 - CT07: Scatto termico
   RUNG wire#powerrail
      Contact( "CT07".Alm.Overload )
      Coil( "Alm".Act.Alm300 )
      Coil( "Alm".Mem.Alm300 )
   END_RUNG
   // the same network as SCL:
   "Alm".Act.Alm300 := "CT07".Alm.Overload;
   "Alm".Mem.Alm300 := "CT07".Alm.Overload;
END_REGION

REGION Network 93: Alm301 - CT08: Scatto termico
   RUNG wire#powerrail
      Contact( "CT08".Alm.Overload )
      Coil( "Alm".Act.Alm301 )
      Coil( "Alm".Mem.Alm301 )
   END_RUNG
   // the same network as SCL:
   "Alm".Act.Alm301 := "CT08".Alm.Overload;
   "Alm".Mem.Alm301 := "CT08".Alm.Overload;
END_REGION

REGION Network 94: Alm302 - CT09: Scatto termico
   RUNG wire#powerrail
      Contact( "CT09".Alm.Overload )
      Coil( "Alm".Act.Alm302 )
      Coil( "Alm".Mem.Alm302 )
   END_RUNG
   // the same network as SCL:
   "Alm".Act.Alm302 := "CT09".Alm.Overload;
   "Alm".Mem.Alm302 := "CT09".Alm.Overload;
END_REGION

REGION Network 95: Alm303 - CT10: Scatto termico
   RUNG wire#powerrail
      Contact( "CT10".Alm.Overload )
      Coil( "Alm".Act.Alm303 )
      Coil( "Alm".Mem.Alm303 )
   END_RUNG
   // the same network as SCL:
   "Alm".Act.Alm303 := "CT10".Alm.Overload;
   "Alm".Mem.Alm303 := "CT10".Alm.Overload;
END_REGION

REGION Network 96: Alm304 - CT11: Scatto termico
   RUNG wire#powerrail
      Contact( "CT11".Alm.Overload )
      Coil( "Alm".Act.Alm304 )
      Coil( "Alm".Mem.Alm304 )
   END_RUNG
   // the same network as SCL:
   "Alm".Act.Alm304 := "CT11".Alm.Overload;
   "Alm".Mem.Alm304 := "CT11".Alm.Overload;
END_REGION

REGION Network 97: Alm305 - CT12: Scatto termico
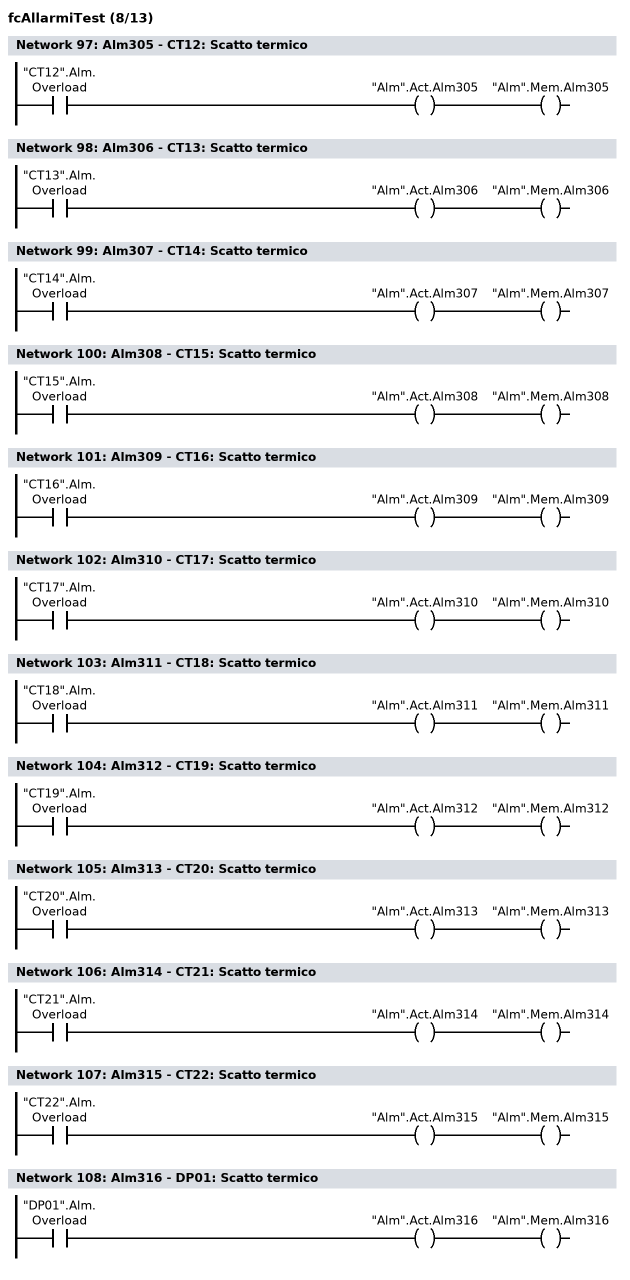
   RUNG wire#powerrail
      Contact( "CT12".Alm.Overload )
      Coil( "Alm".Act.Alm305 )
      Coil( "Alm".Mem.Alm305 )
   END_RUNG
   // the same network as SCL:
   "Alm".Act.Alm305 := "CT12".Alm.Overload;
   "Alm".Mem.Alm305 := "CT12".Alm.Overload;
END_REGION

REGION Network 98: Alm306 - CT13: Scatto termico
   RUNG wire#powerrail
      Contact( "CT13".Alm.Overload )
      Coil( "Alm".Act.Alm306 )
      Coil( "Alm".Mem.Alm306 )
   END_RUNG
   // the same network as SCL:
   "Alm".Act.Alm306 := "CT13".Alm.Overload;
   "Alm".Mem.Alm306 := "CT13".Alm.Overload;
END_REGION

REGION Network 99: Alm307 - CT14: Scatto termico
   RUNG wire#powerrail
      Contact( "CT14".Alm.Overload )
      Coil( "Alm".Act.Alm307 )
      Coil( "Alm".Mem.Alm307 )
   END_RUNG
   // the same network as SCL:
   "Alm".Act.Alm307 := "CT14".Alm.Overload;
   "Alm".Mem.Alm307 := "CT14".Alm.Overload;
END_REGION

REGION Network 100: Alm308 - CT15: Scatto termico
   RUNG wire#powerrail
      Contact( "CT15".Alm.Overload )
      Coil( "Alm".Act.Alm308 )
      Coil( "Alm".Mem.Alm308 )
   END_RUNG
   // the same network as SCL:
   "Alm".Act.Alm308 := "CT15".Alm.Overload;
   "Alm".Mem.Alm308 := "CT15".Alm.Overload;
END_REGION

REGION Network 101: Alm309 - CT16: Scatto termico
   RUNG wire#powerrail
      Contact( "CT16".Alm.Overload )
      Coil( "Alm".Act.Alm309 )
      Coil( "Alm".Mem.Alm309 )
   END_RUNG
   // the same network as SCL:
   "Alm".Act.Alm309 := "CT16".Alm.Overload;
   "Alm".Mem.Alm309 := "CT16".Alm.Overload;
END_REGION

REGION Network 102: Alm310 - CT17: Scatto termico
   RUNG wire#powerrail
      Contact( "CT17".Alm.Overload )
      Coil( "Alm".Act.Alm310 )
      Coil( "Alm".Mem.Alm310 )
   END_RUNG
   // the same network as SCL:
   "Alm".Act.Alm310 := "CT17".Alm.Overload;
   "Alm".Mem.Alm310 := "CT17".Alm.Overload;
END_REGION

REGION Network 103: Alm311 - CT18: Scatto termico
   RUNG wire#powerrail
      Contact( "CT18".Alm.Overload )
      Coil( "Alm".Act.Alm311 )
      Coil( "Alm".Mem.Alm311 )
   END_RUNG
   // the same network as SCL:
   "Alm".Act.Alm311 := "CT18".Alm.Overload;
   "Alm".Mem.Alm311 := "CT18".Alm.Overload;
END_REGION

REGION Network 104: Alm312 - CT19: Scatto termico
   RUNG wire#powerrail
      Contact( "CT19".Alm.Overload )
      Coil( "Alm".Act.Alm312 )
      Coil( "Alm".Mem.Alm312 )
   END_RUNG
   // the same network as SCL:
   "Alm".Act.Alm312 := "CT19".Alm.Overload;
   "Alm".Mem.Alm312 := "CT19".Alm.Overload;
END_REGION

REGION Network 105: Alm313 - CT20: Scatto termico
   RUNG wire#powerrail
      Contact( "CT20".Alm.Overload )
      Coil( "Alm".Act.Alm313 )
      Coil( "Alm".Mem.Alm313 )
   END_RUNG
   // the same network as SCL:
   "Alm".Act.Alm313 := "CT20".Alm.Overload;
   "Alm".Mem.Alm313 := "CT20".Alm.Overload;
END_REGION

REGION Network 106: Alm314 - CT21: Scatto termico
   RUNG wire#powerrail
      Contact( "CT21".Alm.Overload )
      Coil( "Alm".Act.Alm314 )
      Coil( "Alm".Mem.Alm314 )
   END_RUNG
   // the same network as SCL:
   "Alm".Act.Alm314 := "CT21".Alm.Overload;
   "Alm".Mem.Alm314 := "CT21".Alm.Overload;
END_REGION

REGION Network 107: Alm315 - CT22: Scatto termico
   RUNG wire#powerrail
      Contact( "CT22".Alm.Overload )
      Coil( "Alm".Act.Alm315 )
      Coil( "Alm".Mem.Alm315 )
   END_RUNG
   // the same network as SCL:
   "Alm".Act.Alm315 := "CT22".Alm.Overload;
   "Alm".Mem.Alm315 := "CT22".Alm.Overload;
END_REGION

REGION Network 108: Alm316 - DP01: Scatto termico
   RUNG wire#powerrail
      Contact( "DP01".Alm.Overload )
      Coil( "Alm".Act.Alm316 )
      Coil( "Alm".Mem.Alm316 )
   END_RUNG
   // the same network as SCL:
   "Alm".Act.Alm316 := "DP01".Alm.Overload;
   "Alm".Mem.Alm316 := "DP01".Alm.Overload;
END_REGION

REGION Network 109: Alm317 - EFP01: Scatto termico
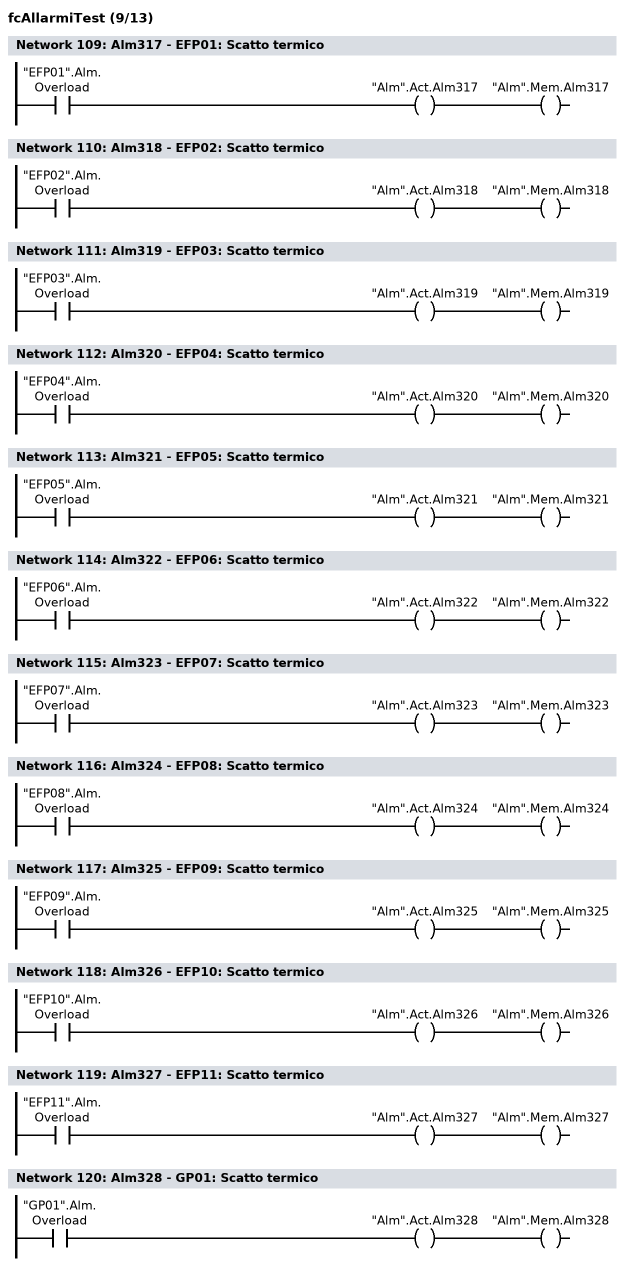
   RUNG wire#powerrail
      Contact( "EFP01".Alm.Overload )
      Coil( "Alm".Act.Alm317 )
      Coil( "Alm".Mem.Alm317 )
   END_RUNG
   // the same network as SCL:
   "Alm".Act.Alm317 := "EFP01".Alm.Overload;
   "Alm".Mem.Alm317 := "EFP01".Alm.Overload;
END_REGION

REGION Network 110: Alm318 - EFP02: Scatto termico
   RUNG wire#powerrail
      Contact( "EFP02".Alm.Overload )
      Coil( "Alm".Act.Alm318 )
      Coil( "Alm".Mem.Alm318 )
   END_RUNG
   // the same network as SCL:
   "Alm".Act.Alm318 := "EFP02".Alm.Overload;
   "Alm".Mem.Alm318 := "EFP02".Alm.Overload;
END_REGION

REGION Network 111: Alm319 - EFP03: Scatto termico
   RUNG wire#powerrail
      Contact( "EFP03".Alm.Overload )
      Coil( "Alm".Act.Alm319 )
      Coil( "Alm".Mem.Alm319 )
   END_RUNG
   // the same network as SCL:
   "Alm".Act.Alm319 := "EFP03".Alm.Overload;
   "Alm".Mem.Alm319 := "EFP03".Alm.Overload;
END_REGION

REGION Network 112: Alm320 - EFP04: Scatto termico
   RUNG wire#powerrail
      Contact( "EFP04".Alm.Overload )
      Coil( "Alm".Act.Alm320 )
      Coil( "Alm".Mem.Alm320 )
   END_RUNG
   // the same network as SCL:
   "Alm".Act.Alm320 := "EFP04".Alm.Overload;
   "Alm".Mem.Alm320 := "EFP04".Alm.Overload;
END_REGION

REGION Network 113: Alm321 - EFP05: Scatto termico
   RUNG wire#powerrail
      Contact( "EFP05".Alm.Overload )
      Coil( "Alm".Act.Alm321 )
      Coil( "Alm".Mem.Alm321 )
   END_RUNG
   // the same network as SCL:
   "Alm".Act.Alm321 := "EFP05".Alm.Overload;
   "Alm".Mem.Alm321 := "EFP05".Alm.Overload;
END_REGION

REGION Network 114: Alm322 - EFP06: Scatto termico
   RUNG wire#powerrail
      Contact( "EFP06".Alm.Overload )
      Coil( "Alm".Act.Alm322 )
      Coil( "Alm".Mem.Alm322 )
   END_RUNG
   // the same network as SCL:
   "Alm".Act.Alm322 := "EFP06".Alm.Overload;
   "Alm".Mem.Alm322 := "EFP06".Alm.Overload;
END_REGION

REGION Network 115: Alm323 - EFP07: Scatto termico
   RUNG wire#powerrail
      Contact( "EFP07".Alm.Overload )
      Coil( "Alm".Act.Alm323 )
      Coil( "Alm".Mem.Alm323 )
   END_RUNG
   // the same network as SCL:
   "Alm".Act.Alm323 := "EFP07".Alm.Overload;
   "Alm".Mem.Alm323 := "EFP07".Alm.Overload;
END_REGION

REGION Network 116: Alm324 - EFP08: Scatto termico
   RUNG wire#powerrail
      Contact( "EFP08".Alm.Overload )
      Coil( "Alm".Act.Alm324 )
      Coil( "Alm".Mem.Alm324 )
   END_RUNG
   // the same network as SCL:
   "Alm".Act.Alm324 := "EFP08".Alm.Overload;
   "Alm".Mem.Alm324 := "EFP08".Alm.Overload;
END_REGION

REGION Network 117: Alm325 - EFP09: Scatto termico
   RUNG wire#powerrail
      Contact( "EFP09".Alm.Overload )
      Coil( "Alm".Act.Alm325 )
      Coil( "Alm".Mem.Alm325 )
   END_RUNG
   // the same network as SCL:
   "Alm".Act.Alm325 := "EFP09".Alm.Overload;
   "Alm".Mem.Alm325 := "EFP09".Alm.Overload;
END_REGION

REGION Network 118: Alm326 - EFP10: Scatto termico
   RUNG wire#powerrail
      Contact( "EFP10".Alm.Overload )
      Coil( "Alm".Act.Alm326 )
      Coil( "Alm".Mem.Alm326 )
   END_RUNG
   // the same network as SCL:
   "Alm".Act.Alm326 := "EFP10".Alm.Overload;
   "Alm".Mem.Alm326 := "EFP10".Alm.Overload;
END_REGION

REGION Network 119: Alm327 - EFP11: Scatto termico
   RUNG wire#powerrail
      Contact( "EFP11".Alm.Overload )
      Coil( "Alm".Act.Alm327 )
      Coil( "Alm".Mem.Alm327 )
   END_RUNG
   // the same network as SCL:
   "Alm".Act.Alm327 := "EFP11".Alm.Overload;
   "Alm".Mem.Alm327 := "EFP11".Alm.Overload;
END_REGION

REGION Network 120: Alm328 - GP01: Scatto termico
   RUNG wire#powerrail
      Contact( "GP01".Alm.Overload )
      Coil( "Alm".Act.Alm328 )
      Coil( "Alm".Mem.Alm328 )
   END_RUNG
   // the same network as SCL:
   "Alm".Act.Alm328 := "GP01".Alm.Overload;
   "Alm".Mem.Alm328 := "GP01".Alm.Overload;
END_REGION

REGION Network 121: Alm329 - GP02: Scatto termico
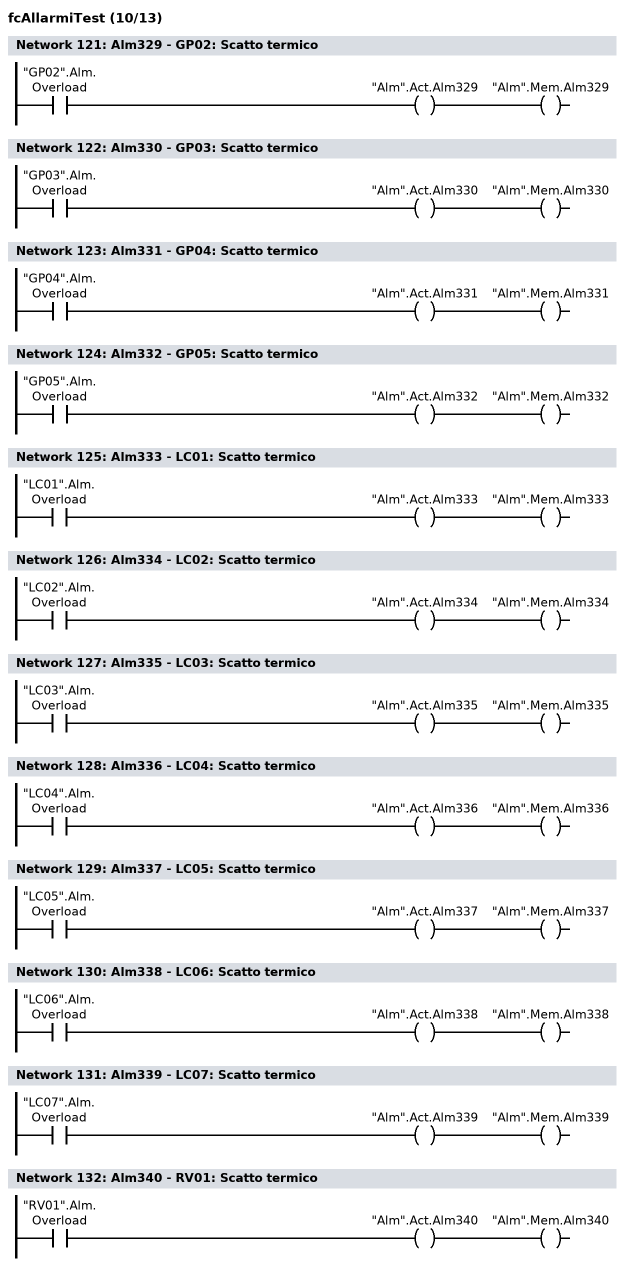
   RUNG wire#powerrail
      Contact( "GP02".Alm.Overload )
      Coil( "Alm".Act.Alm329 )
      Coil( "Alm".Mem.Alm329 )
   END_RUNG
   // the same network as SCL:
   "Alm".Act.Alm329 := "GP02".Alm.Overload;
   "Alm".Mem.Alm329 := "GP02".Alm.Overload;
END_REGION

REGION Network 122: Alm330 - GP03: Scatto termico
   RUNG wire#powerrail
      Contact( "GP03".Alm.Overload )
      Coil( "Alm".Act.Alm330 )
      Coil( "Alm".Mem.Alm330 )
   END_RUNG
   // the same network as SCL:
   "Alm".Act.Alm330 := "GP03".Alm.Overload;
   "Alm".Mem.Alm330 := "GP03".Alm.Overload;
END_REGION

REGION Network 123: Alm331 - GP04: Scatto termico
   RUNG wire#powerrail
      Contact( "GP04".Alm.Overload )
      Coil( "Alm".Act.Alm331 )
      Coil( "Alm".Mem.Alm331 )
   END_RUNG
   // the same network as SCL:
   "Alm".Act.Alm331 := "GP04".Alm.Overload;
   "Alm".Mem.Alm331 := "GP04".Alm.Overload;
END_REGION

REGION Network 124: Alm332 - GP05: Scatto termico
   RUNG wire#powerrail
      Contact( "GP05".Alm.Overload )
      Coil( "Alm".Act.Alm332 )
      Coil( "Alm".Mem.Alm332 )
   END_RUNG
   // the same network as SCL:
   "Alm".Act.Alm332 := "GP05".Alm.Overload;
   "Alm".Mem.Alm332 := "GP05".Alm.Overload;
END_REGION

REGION Network 125: Alm333 - LC01: Scatto termico
   RUNG wire#powerrail
      Contact( "LC01".Alm.Overload )
      Coil( "Alm".Act.Alm333 )
      Coil( "Alm".Mem.Alm333 )
   END_RUNG
   // the same network as SCL:
   "Alm".Act.Alm333 := "LC01".Alm.Overload;
   "Alm".Mem.Alm333 := "LC01".Alm.Overload;
END_REGION

REGION Network 126: Alm334 - LC02: Scatto termico
   RUNG wire#powerrail
      Contact( "LC02".Alm.Overload )
      Coil( "Alm".Act.Alm334 )
      Coil( "Alm".Mem.Alm334 )
   END_RUNG
   // the same network as SCL:
   "Alm".Act.Alm334 := "LC02".Alm.Overload;
   "Alm".Mem.Alm334 := "LC02".Alm.Overload;
END_REGION

REGION Network 127: Alm335 - LC03: Scatto termico
   RUNG wire#powerrail
      Contact( "LC03".Alm.Overload )
      Coil( "Alm".Act.Alm335 )
      Coil( "Alm".Mem.Alm335 )
   END_RUNG
   // the same network as SCL:
   "Alm".Act.Alm335 := "LC03".Alm.Overload;
   "Alm".Mem.Alm335 := "LC03".Alm.Overload;
END_REGION

REGION Network 128: Alm336 - LC04: Scatto termico
   RUNG wire#powerrail
      Contact( "LC04".Alm.Overload )
      Coil( "Alm".Act.Alm336 )
      Coil( "Alm".Mem.Alm336 )
   END_RUNG
   // the same network as SCL:
   "Alm".Act.Alm336 := "LC04".Alm.Overload;
   "Alm".Mem.Alm336 := "LC04".Alm.Overload;
END_REGION

REGION Network 129: Alm337 - LC05: Scatto termico
   RUNG wire#powerrail
      Contact( "LC05".Alm.Overload )
      Coil( "Alm".Act.Alm337 )
      Coil( "Alm".Mem.Alm337 )
   END_RUNG
   // the same network as SCL:
   "Alm".Act.Alm337 := "LC05".Alm.Overload;
   "Alm".Mem.Alm337 := "LC05".Alm.Overload;
END_REGION

REGION Network 130: Alm338 - LC06: Scatto termico
   RUNG wire#powerrail
      Contact( "LC06".Alm.Overload )
      Coil( "Alm".Act.Alm338 )
      Coil( "Alm".Mem.Alm338 )
   END_RUNG
   // the same network as SCL:
   "Alm".Act.Alm338 := "LC06".Alm.Overload;
   "Alm".Mem.Alm338 := "LC06".Alm.Overload;
END_REGION

REGION Network 131: Alm339 - LC07: Scatto termico
   RUNG wire#powerrail
      Contact( "LC07".Alm.Overload )
      Coil( "Alm".Act.Alm339 )
      Coil( "Alm".Mem.Alm339 )
   END_RUNG
   // the same network as SCL:
   "Alm".Act.Alm339 := "LC07".Alm.Overload;
   "Alm".Mem.Alm339 := "LC07".Alm.Overload;
END_REGION

REGION Network 132: Alm340 - RV01: Scatto termico
   RUNG wire#powerrail
      Contact( "RV01".Alm.Overload )
      Coil( "Alm".Act.Alm340 )
      Coil( "Alm".Mem.Alm340 )
   END_RUNG
   // the same network as SCL:
   "Alm".Act.Alm340 := "RV01".Alm.Overload;
   "Alm".Mem.Alm340 := "RV01".Alm.Overload;
END_REGION

REGION Network 133: Alm341 - RV02: Scatto termico
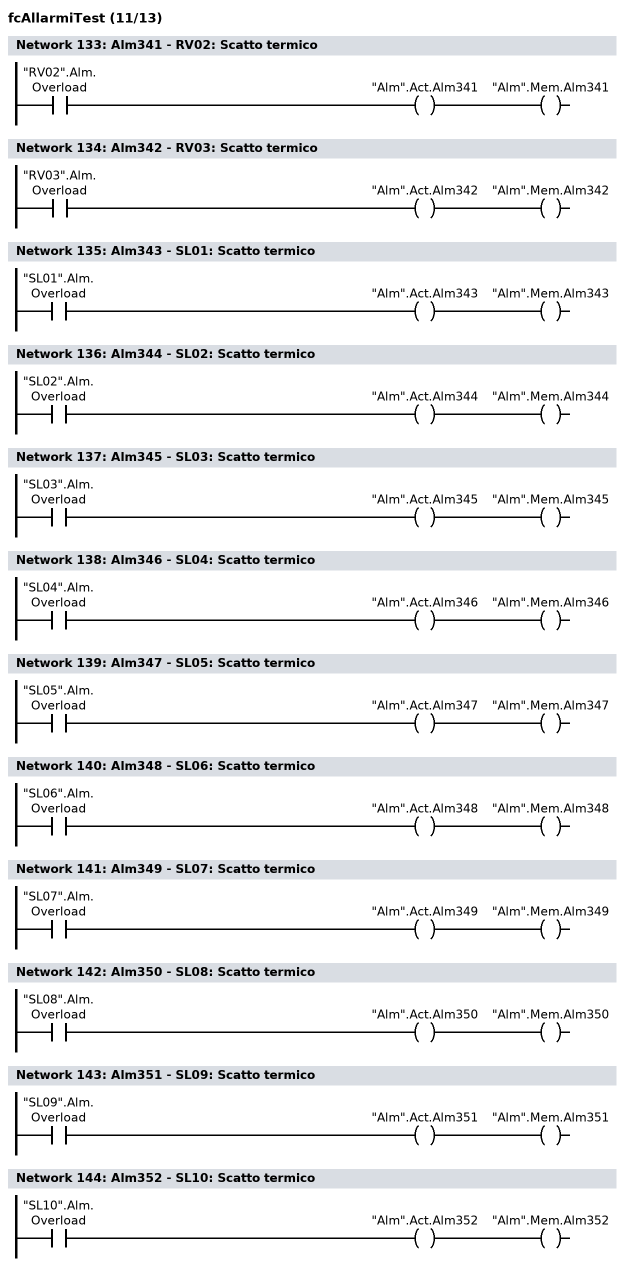
   RUNG wire#powerrail
      Contact( "RV02".Alm.Overload )
      Coil( "Alm".Act.Alm341 )
      Coil( "Alm".Mem.Alm341 )
   END_RUNG
   // the same network as SCL:
   "Alm".Act.Alm341 := "RV02".Alm.Overload;
   "Alm".Mem.Alm341 := "RV02".Alm.Overload;
END_REGION

REGION Network 134: Alm342 - RV03: Scatto termico
   RUNG wire#powerrail
      Contact( "RV03".Alm.Overload )
      Coil( "Alm".Act.Alm342 )
      Coil( "Alm".Mem.Alm342 )
   END_RUNG
   // the same network as SCL:
   "Alm".Act.Alm342 := "RV03".Alm.Overload;
   "Alm".Mem.Alm342 := "RV03".Alm.Overload;
END_REGION

REGION Network 135: Alm343 - SL01: Scatto termico
   RUNG wire#powerrail
      Contact( "SL01".Alm.Overload )
      Coil( "Alm".Act.Alm343 )
      Coil( "Alm".Mem.Alm343 )
   END_RUNG
   // the same network as SCL:
   "Alm".Act.Alm343 := "SL01".Alm.Overload;
   "Alm".Mem.Alm343 := "SL01".Alm.Overload;
END_REGION

REGION Network 136: Alm344 - SL02: Scatto termico
   RUNG wire#powerrail
      Contact( "SL02".Alm.Overload )
      Coil( "Alm".Act.Alm344 )
      Coil( "Alm".Mem.Alm344 )
   END_RUNG
   // the same network as SCL:
   "Alm".Act.Alm344 := "SL02".Alm.Overload;
   "Alm".Mem.Alm344 := "SL02".Alm.Overload;
END_REGION

REGION Network 137: Alm345 - SL03: Scatto termico
   RUNG wire#powerrail
      Contact( "SL03".Alm.Overload )
      Coil( "Alm".Act.Alm345 )
      Coil( "Alm".Mem.Alm345 )
   END_RUNG
   // the same network as SCL:
   "Alm".Act.Alm345 := "SL03".Alm.Overload;
   "Alm".Mem.Alm345 := "SL03".Alm.Overload;
END_REGION

REGION Network 138: Alm346 - SL04: Scatto termico
   RUNG wire#powerrail
      Contact( "SL04".Alm.Overload )
      Coil( "Alm".Act.Alm346 )
      Coil( "Alm".Mem.Alm346 )
   END_RUNG
   // the same network as SCL:
   "Alm".Act.Alm346 := "SL04".Alm.Overload;
   "Alm".Mem.Alm346 := "SL04".Alm.Overload;
END_REGION

REGION Network 139: Alm347 - SL05: Scatto termico
   RUNG wire#powerrail
      Contact( "SL05".Alm.Overload )
      Coil( "Alm".Act.Alm347 )
      Coil( "Alm".Mem.Alm347 )
   END_RUNG
   // the same network as SCL:
   "Alm".Act.Alm347 := "SL05".Alm.Overload;
   "Alm".Mem.Alm347 := "SL05".Alm.Overload;
END_REGION

REGION Network 140: Alm348 - SL06: Scatto termico
   RUNG wire#powerrail
      Contact( "SL06".Alm.Overload )
      Coil( "Alm".Act.Alm348 )
      Coil( "Alm".Mem.Alm348 )
   END_RUNG
   // the same network as SCL:
   "Alm".Act.Alm348 := "SL06".Alm.Overload;
   "Alm".Mem.Alm348 := "SL06".Alm.Overload;
END_REGION

REGION Network 141: Alm349 - SL07: Scatto termico
   RUNG wire#powerrail
      Contact( "SL07".Alm.Overload )
      Coil( "Alm".Act.Alm349 )
      Coil( "Alm".Mem.Alm349 )
   END_RUNG
   // the same network as SCL:
   "Alm".Act.Alm349 := "SL07".Alm.Overload;
   "Alm".Mem.Alm349 := "SL07".Alm.Overload;
END_REGION

REGION Network 142: Alm350 - SL08: Scatto termico
   RUNG wire#powerrail
      Contact( "SL08".Alm.Overload )
      Coil( "Alm".Act.Alm350 )
      Coil( "Alm".Mem.Alm350 )
   END_RUNG
   // the same network as SCL:
   "Alm".Act.Alm350 := "SL08".Alm.Overload;
   "Alm".Mem.Alm350 := "SL08".Alm.Overload;
END_REGION

REGION Network 143: Alm351 - SL09: Scatto termico
   RUNG wire#powerrail
      Contact( "SL09".Alm.Overload )
      Coil( "Alm".Act.Alm351 )
      Coil( "Alm".Mem.Alm351 )
   END_RUNG
   // the same network as SCL:
   "Alm".Act.Alm351 := "SL09".Alm.Overload;
   "Alm".Mem.Alm351 := "SL09".Alm.Overload;
END_REGION

REGION Network 144: Alm352 - SL10: Scatto termico
   RUNG wire#powerrail
      Contact( "SL10".Alm.Overload )
      Coil( "Alm".Act.Alm352 )
      Coil( "Alm".Mem.Alm352 )
   END_RUNG
   // the same network as SCL:
   "Alm".Act.Alm352 := "SL10".Alm.Overload;
   "Alm".Mem.Alm352 := "SL10".Alm.Overload;
END_REGION

REGION Network 145: Alm353 - SL11: Scatto termico
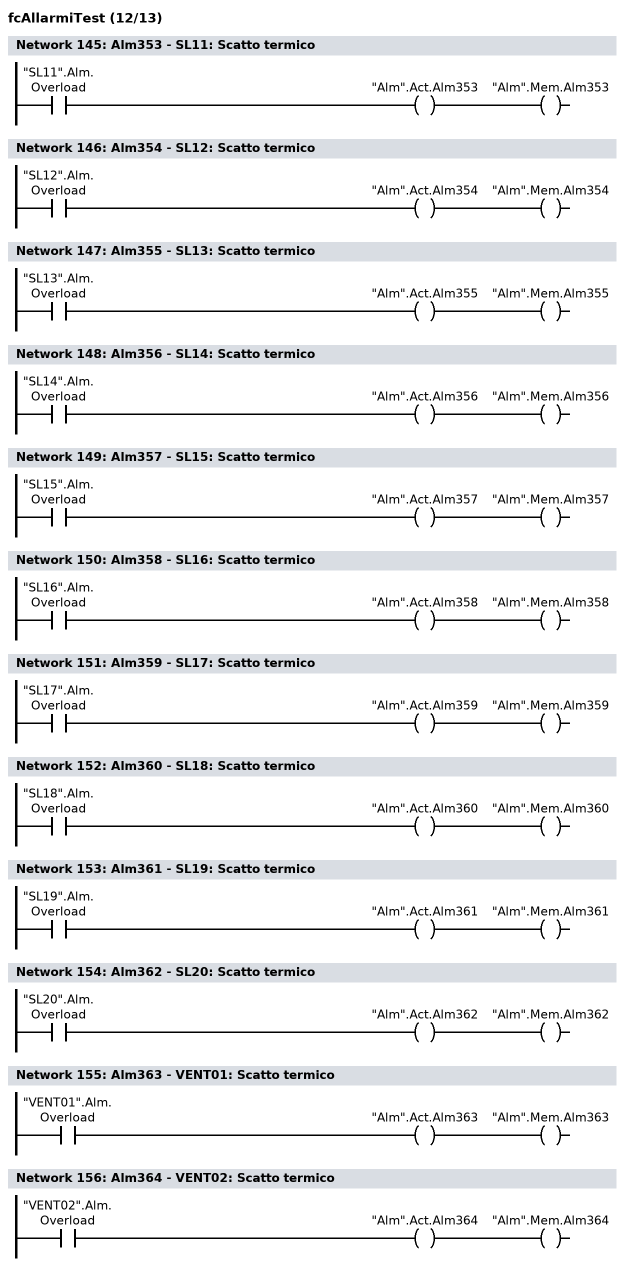
   RUNG wire#powerrail
      Contact( "SL11".Alm.Overload )
      Coil( "Alm".Act.Alm353 )
      Coil( "Alm".Mem.Alm353 )
   END_RUNG
   // the same network as SCL:
   "Alm".Act.Alm353 := "SL11".Alm.Overload;
   "Alm".Mem.Alm353 := "SL11".Alm.Overload;
END_REGION

REGION Network 146: Alm354 - SL12: Scatto termico
   RUNG wire#powerrail
      Contact( "SL12".Alm.Overload )
      Coil( "Alm".Act.Alm354 )
      Coil( "Alm".Mem.Alm354 )
   END_RUNG
   // the same network as SCL:
   "Alm".Act.Alm354 := "SL12".Alm.Overload;
   "Alm".Mem.Alm354 := "SL12".Alm.Overload;
END_REGION

REGION Network 147: Alm355 - SL13: Scatto termico
   RUNG wire#powerrail
      Contact( "SL13".Alm.Overload )
      Coil( "Alm".Act.Alm355 )
      Coil( "Alm".Mem.Alm355 )
   END_RUNG
   // the same network as SCL:
   "Alm".Act.Alm355 := "SL13".Alm.Overload;
   "Alm".Mem.Alm355 := "SL13".Alm.Overload;
END_REGION

REGION Network 148: Alm356 - SL14: Scatto termico
   RUNG wire#powerrail
      Contact( "SL14".Alm.Overload )
      Coil( "Alm".Act.Alm356 )
      Coil( "Alm".Mem.Alm356 )
   END_RUNG
   // the same network as SCL:
   "Alm".Act.Alm356 := "SL14".Alm.Overload;
   "Alm".Mem.Alm356 := "SL14".Alm.Overload;
END_REGION

REGION Network 149: Alm357 - SL15: Scatto termico
   RUNG wire#powerrail
      Contact( "SL15".Alm.Overload )
      Coil( "Alm".Act.Alm357 )
      Coil( "Alm".Mem.Alm357 )
   END_RUNG
   // the same network as SCL:
   "Alm".Act.Alm357 := "SL15".Alm.Overload;
   "Alm".Mem.Alm357 := "SL15".Alm.Overload;
END_REGION

REGION Network 150: Alm358 - SL16: Scatto termico
   RUNG wire#powerrail
      Contact( "SL16".Alm.Overload )
      Coil( "Alm".Act.Alm358 )
      Coil( "Alm".Mem.Alm358 )
   END_RUNG
   // the same network as SCL:
   "Alm".Act.Alm358 := "SL16".Alm.Overload;
   "Alm".Mem.Alm358 := "SL16".Alm.Overload;
END_REGION

REGION Network 151: Alm359 - SL17: Scatto termico
   RUNG wire#powerrail
      Contact( "SL17".Alm.Overload )
      Coil( "Alm".Act.Alm359 )
      Coil( "Alm".Mem.Alm359 )
   END_RUNG
   // the same network as SCL:
   "Alm".Act.Alm359 := "SL17".Alm.Overload;
   "Alm".Mem.Alm359 := "SL17".Alm.Overload;
END_REGION

REGION Network 152: Alm360 - SL18: Scatto termico
   RUNG wire#powerrail
      Contact( "SL18".Alm.Overload )
      Coil( "Alm".Act.Alm360 )
      Coil( "Alm".Mem.Alm360 )
   END_RUNG
   // the same network as SCL:
   "Alm".Act.Alm360 := "SL18".Alm.Overload;
   "Alm".Mem.Alm360 := "SL18".Alm.Overload;
END_REGION

REGION Network 153: Alm361 - SL19: Scatto termico
   RUNG wire#powerrail
      Contact( "SL19".Alm.Overload )
      Coil( "Alm".Act.Alm361 )
      Coil( "Alm".Mem.Alm361 )
   END_RUNG
   // the same network as SCL:
   "Alm".Act.Alm361 := "SL19".Alm.Overload;
   "Alm".Mem.Alm361 := "SL19".Alm.Overload;
END_REGION

REGION Network 154: Alm362 - SL20: Scatto termico
   RUNG wire#powerrail
      Contact( "SL20".Alm.Overload )
      Coil( "Alm".Act.Alm362 )
      Coil( "Alm".Mem.Alm362 )
   END_RUNG
   // the same network as SCL:
   "Alm".Act.Alm362 := "SL20".Alm.Overload;
   "Alm".Mem.Alm362 := "SL20".Alm.Overload;
END_REGION

REGION Network 155: Alm363 - VENT01: Scatto termico
   RUNG wire#powerrail
      Contact( "VENT01".Alm.Overload )
      Coil( "Alm".Act.Alm363 )
      Coil( "Alm".Mem.Alm363 )
   END_RUNG
   // the same network as SCL:
   "Alm".Act.Alm363 := "VENT01".Alm.Overload;
   "Alm".Mem.Alm363 := "VENT01".Alm.Overload;
END_REGION

REGION Network 156: Alm364 - VENT02: Scatto termico
   RUNG wire#powerrail
      Contact( "VENT02".Alm.Overload )
      Coil( "Alm".Act.Alm364 )
      Coil( "Alm".Mem.Alm364 )
   END_RUNG
   // the same network as SCL:
   "Alm".Act.Alm364 := "VENT02".Alm.Overload;
   "Alm".Mem.Alm364 := "VENT02".Alm.Overload;
END_REGION

REGION Network 157: Alm365 - VENT03: Scatto termico
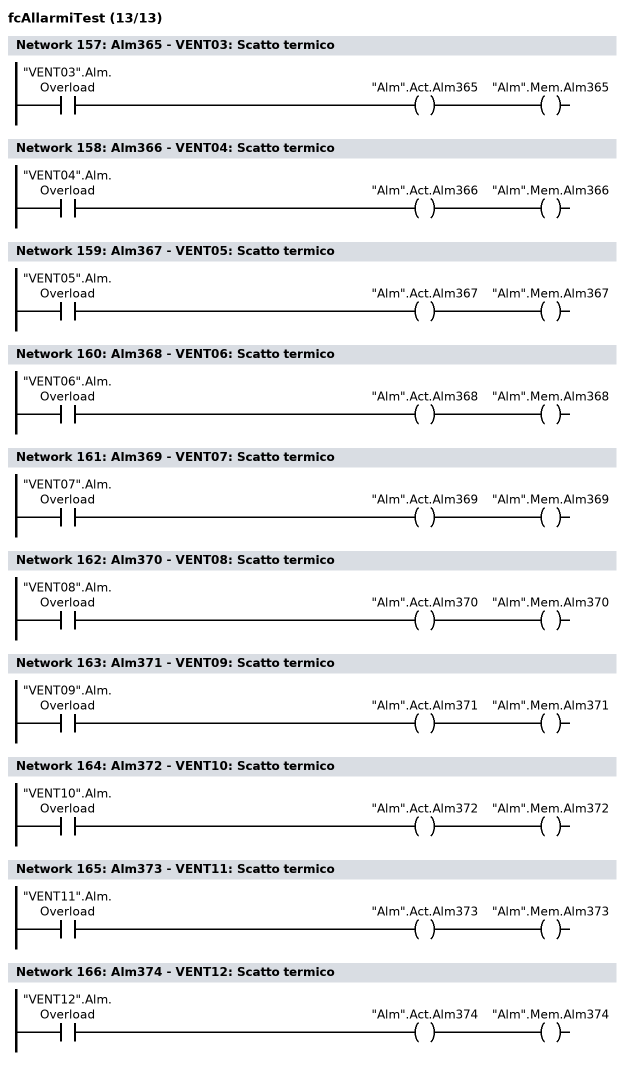
   RUNG wire#powerrail
      Contact( "VENT03".Alm.Overload )
      Coil( "Alm".Act.Alm365 )
      Coil( "Alm".Mem.Alm365 )
   END_RUNG
   // the same network as SCL:
   "Alm".Act.Alm365 := "VENT03".Alm.Overload;
   "Alm".Mem.Alm365 := "VENT03".Alm.Overload;
END_REGION

REGION Network 158: Alm366 - VENT04: Scatto termico
   RUNG wire#powerrail
      Contact( "VENT04".Alm.Overload )
      Coil( "Alm".Act.Alm366 )
      Coil( "Alm".Mem.Alm366 )
   END_RUNG
   // the same network as SCL:
   "Alm".Act.Alm366 := "VENT04".Alm.Overload;
   "Alm".Mem.Alm366 := "VENT04".Alm.Overload;
END_REGION

REGION Network 159: Alm367 - VENT05: Scatto termico
   RUNG wire#powerrail
      Contact( "VENT05".Alm.Overload )
      Coil( "Alm".Act.Alm367 )
      Coil( "Alm".Mem.Alm367 )
   END_RUNG
   // the same network as SCL:
   "Alm".Act.Alm367 := "VENT05".Alm.Overload;
   "Alm".Mem.Alm367 := "VENT05".Alm.Overload;
END_REGION

REGION Network 160: Alm368 - VENT06: Scatto termico
   RUNG wire#powerrail
      Contact( "VENT06".Alm.Overload )
      Coil( "Alm".Act.Alm368 )
      Coil( "Alm".Mem.Alm368 )
   END_RUNG
   // the same network as SCL:
   "Alm".Act.Alm368 := "VENT06".Alm.Overload;
   "Alm".Mem.Alm368 := "VENT06".Alm.Overload;
END_REGION

REGION Network 161: Alm369 - VENT07: Scatto termico
   RUNG wire#powerrail
      Contact( "VENT07".Alm.Overload )
      Coil( "Alm".Act.Alm369 )
      Coil( "Alm".Mem.Alm369 )
   END_RUNG
   // the same network as SCL:
   "Alm".Act.Alm369 := "VENT07".Alm.Overload;
   "Alm".Mem.Alm369 := "VENT07".Alm.Overload;
END_REGION

REGION Network 162: Alm370 - VENT08: Scatto termico
   RUNG wire#powerrail
      Contact( "VENT08".Alm.Overload )
      Coil( "Alm".Act.Alm370 )
      Coil( "Alm".Mem.Alm370 )
   END_RUNG
   // the same network as SCL:
   "Alm".Act.Alm370 := "VENT08".Alm.Overload;
   "Alm".Mem.Alm370 := "VENT08".Alm.Overload;
END_REGION

REGION Network 163: Alm371 - VENT09: Scatto termico
   RUNG wire#powerrail
      Contact( "VENT09".Alm.Overload )
      Coil( "Alm".Act.Alm371 )
      Coil( "Alm".Mem.Alm371 )
   END_RUNG
   // the same network as SCL:
   "Alm".Act.Alm371 := "VENT09".Alm.Overload;
   "Alm".Mem.Alm371 := "VENT09".Alm.Overload;
END_REGION

REGION Network 164: Alm372 - VENT10: Scatto termico
   RUNG wire#powerrail
      Contact( "VENT10".Alm.Overload )
      Coil( "Alm".Act.Alm372 )
      Coil( "Alm".Mem.Alm372 )
   END_RUNG
   // the same network as SCL:
   "Alm".Act.Alm372 := "VENT10".Alm.Overload;
   "Alm".Mem.Alm372 := "VENT10".Alm.Overload;
END_REGION

REGION Network 165: Alm373 - VENT11: Scatto termico
   RUNG wire#powerrail
      Contact( "VENT11".Alm.Overload )
      Coil( "Alm".Act.Alm373 )
      Coil( "Alm".Mem.Alm373 )
   END_RUNG
   // the same network as SCL:
   "Alm".Act.Alm373 := "VENT11".Alm.Overload;
   "Alm".Mem.Alm373 := "VENT11".Alm.Overload;
END_REGION

REGION Network 166: Alm374 - VENT12: Scatto termico
   RUNG wire#powerrail
      Contact( "VENT12".Alm.Overload )
      Coil( "Alm".Act.Alm374 )
      Coil( "Alm".Mem.Alm374 )
   END_RUNG
   // the same network as SCL:
   "Alm".Act.Alm374 := "VENT12".Alm.Overload;
   "Alm".Mem.Alm374 := "VENT12".Alm.Overload;
END_REGION
END_FUNCTION
